(* PLC project EPEC_CU2.project, CODESYS V3.5 SP19, author XXXX *)
(* stored: creationDateTime 2026-03-19T14:01:24.5297586+02:00, modificationDateTime 2026-03-19T14:01:24.5297586+02:00, organization XXXX *)

(* NOTE! NOTE! NOTE! NOTE! NOTE! NOTE! NOTE! NOTE! NOTE! NOTE! NOTE! This object is created by Epec MultiTool. User changes are overwritten when project is imported. Content: - EventCode channel IDs *)
{attribute 'qualified_only'}
{attribute 'strict'}
TYPE ChannelIDs : (Ch1 := 0, Ch2, Ch3, Ch4) BYTE;
END_TYPE

(* NOTE! NOTE! NOTE! NOTE! NOTE! NOTE! NOTE! NOTE! NOTE! NOTE! NOTE! This object is created by Epec MultiTool. User changes are overwritten when project is imported. Content: - EventCode device IDs *)
{attribute 'qualified_only'}
{attribute 'strict'}
TYPE DeviceIDs : (VoltageInput := 0, DigitalInput, CurrentInput, ParameterValidation) BYTE;
END_TYPE

TYPE IdentityObject : STRUCT
  VendorId : DWORD := 0;  (* Vendor ID *)
  ProductCode : DWORD := 0;  (* Product code *)
  Revision : DWORD := 0;  (* Revision number *)
  SerialNumber : DWORD := 0;  (* Serial number for control unit *)
END_STRUCT;
END_TYPE

{attribute 'qualified_only'}
{attribute 'location' := '16#800'}
{attribute 'strict'}
TYPE InitCanProtocolStates : (INIT_CANOPEN_PROTOCOLS := 1, INIT_CANOPEN_OD := 2, INIT_CANOPEN_PDO := 3, INIT_CANOPEN_OD_SAVE := 4, INIT_CANOPEN_OD_REORG := 5, INIT_J1939 := 6, INIT_PROTOCOLS_DONE := 7);
END_TYPE

TYPE IdentityObject : STRUCT
  VendorId : DWORD := 0;  (* Vendor ID *)
  ProductCode : DWORD := 0;  (* Product code *)
  Revision : DWORD := 0;  (* Revision number *)
  SerialNumber : DWORD := 0;  (* Serial number for control unit *)
END_STRUCT;
END_TYPE

{attribute 'analysis' := '-43'}
VAR_GLOBAL CONSTANT  (* G_CONSTANTS - NOTE! NOTE! NOTE! NOTE! NOTE! NOTE! NOTE! NOTE! NOTE! NOTE! NOTE! This object is created by Epec MultiTool. User changes are overwritten when project is imported. Content: - Project specific constant definitions *)
  DIAG_MCU_TEMP_HIGH_LIMIT : DINT := 125;  (* Diagnostic limit constants *)
  DIAG_MCU_TEMP_LOW_LIMIT : DINT := -40;
  DIAG_MCU_TEMP_DELAY : UINT := 50;
  DIAG_PCB1_TEMP_HIGH_LIMIT : DINT := 125;
  DIAG_PCB1_TEMP_LOW_LIMIT : DINT := -45;
  DIAG_PCB1_TEMP_DELAY : UINT := 100;
  DIAG_PCB2_TEMP_HIGH_LIMIT : DINT := 105;
  DIAG_PCB2_TEMP_LOW_LIMIT : DINT := -40;
  DIAG_PCB2_TEMP_DELAY : UINT := 100;
  DIAG_SUPPLY_VOLTAGE_HIGH_LIMIT : DINT := 32000;
  DIAG_SUPPLY_VOLTAGE_LOW_LIMIT : DINT := 4500;
  DIAG_SUPPLY_VOLTAGE_DELAY : UINT := 450;
  DIAG_OUTPUT_GROUP1_HIGH_LIMIT : DINT := 37000;
  DIAG_OUTPUT_GROUP1_LOW_LIMIT : DINT := 4500;
  DIAG_OUTPUT_GROUP1_DELAY : UINT := 100;
  G_PARAMHANDLERKEYWORD : DWORD := 16#226D6F52;  (* Parameterhandler keyword *)
  G_PARAMETER_SAVE_STATUS_ERROR : BYTE := BYTE#16#00;
  G_PARAMETER_SAVE_STATUS_DONE : BYTE := BYTE#16#01;
  G_PARAMETER_SAVE_STATUS_IN_PROGRESS : BYTE := BYTE#16#FF;
  G_SAFE_PARAMETERS_AUTHENTICATED : BYTE := BYTE#1;
  G_SAFE_PARAMETERS_NOT_AUTHENTICATED : BYTE := BYTE#0;
END_VAR

{attribute 'qualified_only'}
VAR_GLOBAL  (* G_CAN - NOTE! NOTE! NOTE! NOTE! NOTE! NOTE! NOTE! NOTE! NOTE! NOTE! NOTE! This object is created by Epec MultiTool. User changes are overwritten when project is imported. Content: - CAN definitions *)
  Channel1 : EPEC_CANL2.Channel;
  Channel2 : EPEC_CANL2.Channel;
  Channel3 : EPEC_CANL2.Channel;
  Channel4 : EPEC_CANL2.Channel;
  Channel5 : EPEC_CANL2.Channel;
  Channel6 : EPEC_CANL2.Channel;
END_VAR

{attribute 'qualified_only'}
{attribute 'location' := '16#800'}
{attribute 'analysis' := '-6, -12, -33, -43'}
VAR_GLOBAL  (* G_Common *)
  ParHandler : EPEC_PH.ParameterHandler;  (* Parameterhandler. Utility library for ODSave. Library handles parameter image modification. *)
  ParameterArea : ARRAY[1..EPEC_HWD.LibParameters.G_PARAM_AREA_MAX_SIZE] OF BYTE;  (* Parameter image *)
  FastParHandler : EPEC_PH.ParameterHandler;
  FastParameterArea : ARRAY[1..EPEC_HWD.LibParameters.G_USER_VALUE_AREA_MAX_SIZE] OF BYTE;
  FastParameters : FastParameters;
  SaveFastParameters : BOOL := FALSE;
  ParhandlerDisableChanges : BOOL := FALSE;  (* Flag to call Parhandler.DisableChanges(TRUE) *)
  ParhandlerEnableChanges : BOOL := FALSE;  (* Flag to call Parhandler.DisableChanges(FALSE) *)
  CAN1SSDOHandlerGrantAccess : BOOL := FALSE;  (* Flag to call G_CANopen_CAN1.SSDO_Handler.GrantAccessToSafetyParameters(TRUE) *)
  CAN2SSDOHandlerGrantAccess : BOOL := FALSE;  (* Flag to call G_CANopen_CAN2.SSDO_Handler.GrantAccessToSafetyParameters(TRUE) *)
  CAN3SSDOHandlerGrantAccess : BOOL := FALSE;  (* Flag to call G_CANopen_CAN3.SSDO_Handler.GrantAccessToSafetyParameters(TRUE) *)
  CAN4SSDOHandlerGrantAccess : BOOL := FALSE;  (* Flag to call G_CANopen_CAN4.SSDO_Handler.GrantAccessToSafetyParameters(TRUE) *)
  CAN5SSDOHandlerGrantAccess : BOOL := FALSE;  (* Flag to call G_CANopen_CAN5.SSDO_Handler.GrantAccessToSafetyParameters(TRUE) *)
  CAN6SSDOHandlerGrantAccess : BOOL := FALSE;  (* Flag to call G_CANopen_CAN6.SSDO_Handler.GrantAccessToSafetyParameters(TRUE) *)
  ProjectKey : STRING(79) := 'KEeJGzzvbvqAy4c';  (* Project key, used for validating the response code *)
END_VAR


{attribute 'qualified_only'}
{attribute 'location' := '16#800'}
{attribute 'analysis' := '-6'}
VAR_GLOBAL  (* G_Logs *)
  ApplicationLog : EPEC_SERRLOG.ErrorLog;
  AppLogInitOK : BOOL;
END_VAR


{attribute 'qualified_only'}
{attribute 'location' := '16#800'}
{attribute 'analysis' := '-12, -33, -43'}
VAR_GLOBAL  (* G_StatusFlags - NOTE! NOTE! NOTE! NOTE! NOTE! NOTE! NOTE! NOTE! NOTE! NOTE! NOTE! This object is created by Epec MultiTool. User changes are overwritten when project is imported. Content: - PLC_PRG status flags *)
  CANopenCan1NMTResetRequest : BOOL := FALSE;  (* Reset request flags tell if module is wanted to reset after current application cycle. *)
  CANopenCan2NMTResetRequest : BOOL := FALSE;
  CANopenCan3NMTResetRequest : BOOL := FALSE;
  CANopenCan4NMTResetRequest : BOOL := FALSE;
  CANopenCan5NMTResetRequest : BOOL := FALSE;
  CANopenCan6NMTResetRequest : BOOL := FALSE;
  SystemOk : BOOL := FALSE;
  CustomLEDControlEnable : BOOL := FALSE;  (* Flags to control the status LED from the application *)
  RedLED : BOOL := FALSE;
  GreenLED : BOOL := FALSE;
  BlueLED : BOOL := FALSE;
  CustomLED2ControlEnable : BOOL := FALSE;  (* Flags to control the status LED 2 from the application *)
  RedLED2 : BOOL := FALSE;
  GreenLED2 : BOOL := FALSE;
  BlueLED2 : BOOL := FALSE;
END_VAR

{attribute 'qualified_only'}
VAR_GLOBAL  (* G_StatusFlags_Safe - NOTE! NOTE! NOTE! NOTE! NOTE! NOTE! NOTE! NOTE! NOTE! NOTE! NOTE! This object is created by Epec MultiTool. User changes are overwritten when project is imported. Content: - S_PLC_PRG status flags *)
  S_SafeOperationEnable : SAFEBOOL := FALSE;
END_VAR

{attribute 'qualified_only'}
{attribute 'location' := '16#800'}
{attribute 'analysis' := '-33, -43'}
VAR_GLOBAL  (* G_SystemInfo - NOTE! NOTE! NOTE! NOTE! NOTE! NOTE! NOTE! NOTE! NOTE! NOTE! NOTE! This object is created by Epec MultiTool. User changes are overwritten when project is imported. Content: - System information common for all ODs. *)
  ProjectInfo : PROJECT_INFO;
  DeviceName : STRING(79);  (* 16#1008: Manufacturer device name *)
  HWVersion : STRING(79);  (* 16#1009: Manufacturer hardware version *)
  SWVersion : STRING(79);  (* 16#100A: Manufacturer software version *)
  Identity : IdentityObject;  (* 16#1018: Identity object *)
  ToolsVersion : ARRAY[1..1] OF DWORD;  (* 16#2030 Codesys version *)
  WireHarnessId : ARRAY[1..30] OF WORD := [30(0)];  (* 16#2101 Wire harness Sub1: Wire harness ID enable Sub2: Wire harness ID internal adc config Sub3: Wire harness ID internal adc config Sub4: Wire harness ID internal adc config Sub5: Wire harness ID internal adc config Sub6: Wire harness ID internal adc config Sub7: Wire harness ID internal adc config Sub8: Wire harness ID internal adc config Sub9: Wire harness ID internal adc config Sub10: Wire harness ID internal adc config Sub11: Wire harness ID internal adc config Sub12: Wire harness ID internal adc config Sub13: Wire harness ID internal adc config Sub14: Wire harness ID internal adc config Sub15: Wire harness ID internal adc config Sub16: Wire harness ID internal adc config Sub17: Wire harness ID internal adc config Sub18: Wire harness ID internal adc config Sub19: Wire harness ID internal adc config Sub20: Wire harness ID internal adc config Sub21: Wire harness ID internal adc config Sub22: Wire harness ID internal adc config Sub23: Wire harness ID internal adc config Sub24: Wire harness ID internal adc config Sub25: Wire harness ID internal adc config Sub26: Wire harness ID default base offset Sub27: Wire harness ID calculated offset Sub28: Wire harness ID stored offset Sub29: Wire harness ID locked Sub30: Wire harness ID error *)
  SoftwareInformation : ARRAY[1..10] OF STRING(79) := [''];  (* 16#2130 Software information Sub1: Application version Sub2: Additional version information Sub3: Reserved for future use Sub4: Reserved for future use Sub5: Reserved for future use Sub6: Reserved for future use Sub7: Reserved for future use Sub8: Reserved for future use Sub9: Reserved for future use Sub10: Reserved for future use *)
  MACAddress : ARRAY[1..6] OF BYTE := [6(0)];  (* 16#2140 MAC address Sub1: MAC address byte 1 Sub2: MAC address byte 2 Sub3: MAC address byte 3 Sub4: MAC address byte 4 Sub5: MAC address byte 5 Sub6: MAC address byte 6 *)
  EthernetConfiguration : ARRAY[1..50] OF BYTE := [50(0)];  (* 16#2141 Ethernet configuration Sub1: Ethernet enabled/disabled Sub2: DHCP on/off Sub3: Reserved Sub4: Reserved Sub5: Reserved Sub6: Reserved Sub7: Reserved Sub8: Reserved Sub9: Reserved Sub10: Reserved Sub11: Reserved Sub12: Reserved Sub13: Reserved Sub14: Reserved Sub15: Reserved Sub16: Reserved Sub17: Reserved Sub18: Netstatus Sub19: IP address highest byte Sub20: IP address 3rd byte Sub21: IP address 2nd byte Sub22: IP address lowest byte Sub23: Gateway highest byte Sub24: Gateway 3rd byte Sub25: Gateway 2nd byte Sub26: Gateway lowest byte Sub27: Netmask highest byte Sub28: Netmask 3rd byte Sub29: Netmask 2nd byte Sub30: Netmask first byte Sub31: Reserved Sub32: Reserved Sub33: Reserved Sub34: Reserved Sub35: Reserved Sub36: Reserved Sub37: Reserved Sub38: Reserved Sub39: Reserved Sub40: Reserved Sub41: Reserved Sub42: Reserved Sub43: Reserved Sub44: Reserved Sub45: Reserved Sub46: Reserved Sub47: Reserved Sub48: Reserved Sub49: Reserved Sub50: Reserved *)
  CAN1_Comms : ARRAY[1..10] OF WORD := [10(0)];  (* 16#2150 CAN 1 Communication parameters Sub1: CODESYS communication enabled Sub2: CODESYS communication node-ID Sub3: Bit rate Sub4: Cable detection offset for CODESYS node-ID Sub5: Cable detection offset for PLCopen node-ID Sub6: Mask for cable detection pins Sub7: Reserved Sub8: Reserved Sub9: Reserved Sub10: PLCopen application node-ID in CAN1 *)
  CAN2_Comms : ARRAY[1..10] OF WORD := [10(0)];  (* 16#2151 CAN 2 Communication parameters Sub1: CODESYS communication enabled Sub2: CODESYS communication node-ID Sub3: Bit rate Sub4: Reserved Sub5: Reserved Sub6: Reserved Sub7: Reserved Sub8: Reserved Sub9: Reserved Sub10: PLCopen application node-ID in CAN2 *)
  CAN3_Comms : ARRAY[1..10] OF WORD := [10(0)];  (* 16#2152 CAN 3 Communication parameters Sub1: CODESYS communication enabled Sub2: CODESYS communication node-ID Sub3: Bit rate Sub4: Reserved Sub5: Reserved Sub6: Reserved Sub7: Reserved Sub8: Reserved Sub9: Reserved Sub10: PLCopen application node-ID in CAN3 *)
  CAN4_Comms : ARRAY[1..10] OF WORD := [10(0)];  (* 16#2153 CAN 4 Communication parameters Sub1: CODESYS communication enabled Sub2: CODESYS communication node-ID Sub3: Bit rate Sub4: Reserved Sub5: Reserved Sub6: Reserved Sub7: Reserved Sub8: Reserved Sub9: Reserved Sub10: PLCopen application node-ID in CAN4 *)
  CAN5_Comms : ARRAY[1..10] OF WORD := [10(0)];  (* 16#2154 CAN 5 Communication parameters Sub1: CODESYS communication enabled Sub2: CODESYS communication node-ID Sub3: Bit rate Sub4: Reserved Sub5: Reserved Sub6: Reserved Sub7: Reserved Sub8: Reserved Sub9: Reserved Sub10: PLCopen application node-ID in CAN5 *)
  CAN6_Comms : ARRAY[1..10] OF WORD := [10(0)];  (* 16#2155 CAN 6 Communication parameters Sub1: CODESYS communication enabled Sub2: CODESYS communication node-ID Sub3: Bit rate Sub4: Reserved Sub5: Reserved Sub6: Reserved Sub7: Reserved Sub8: Reserved Sub9: Reserved Sub10: PLCopen application node-ID in CAN6 *)
END_VAR

{attribute 'qualified_only'}
{attribute 'global_init_slot' := '49991'}
VAR_GLOBAL  (* G_CANopen_CAN1 - NOTE! NOTE! NOTE! NOTE! NOTE! NOTE! NOTE! NOTE! NOTE! NOTE! NOTE! This object is created by Epec MultiTool User changes are overwritten when project is imported Content - CANopen protocol variable definitions *)
  Device : EPEC_CANopen.Device;  (* CAN device *)
  OD : EPEC_CANopen.OD;  (* Object Dictionary data *)
  ODEntrys : ARRAY[1..86] OF EPEC_CANopen.ODEntry;
  Protocols : ARRAY[1..5] OF EPEC_CANopen.ProtocolEntry;  (* Protocol data *)
  HB : EPEC_CANopen.HBData;  (* Heartbeat producer/consumer protocol data *)
  HB_Handler : EPEC_CANopen.CANopenHB;  (* Heartbeat producer/consumer protocol handler *)
  NMT : EPEC_CANopen.NMTData;  (* NMT protocol data *)
  NMT_Handler : EPEC_CANopen.CANopenNMT;  (* NMT protocol handler *)
  SSDO : EPEC_CANopen.SSDOData;  (* SDO server protocol data *)
  SSDO_Handler : EPEC_CANopen.CANopenSDOServer;  (* SDO server protocol handler *)
  GFC : EPEC_CANopen.GFCData;  (* GFC protocol data *)
  GFC_Handler : EPEC_CANopen.CANopenGFC;  (* GFC protocol handler *)
  CSDOS : ARRAY[1..1] OF EPEC_CANopen.CANopenCSDO := [];  (* SDO client instances *)
  ConfigurationValidCallback : EPEC_CANopen.CallbackOfIndex13FEh;  (* 16#13FE Configuration valid *)
  AppLogDomain : EPEC_CANopen.Domain;  (* 16#2171 Application log domain *)
  SaveAll : EPEC_ODSave.SaveODSaveAll;
  DeleteAll : EPEC_ODSave.SaveODDeleteAll;
  SaveODHandler : EPEC_ODSave.SaveOD_Handler;
  SaveData : ARRAY[0..3] OF EPEC_ODSave.SaveODSubIndexDescription := [(StartIndex := 16#1000, EndIndex := 16#FFFF, GroupNum := 1), (StartIndex := 16#1000, EndIndex := 16#1FFF, GroupNum := 1), (StartIndex := 16#2000, EndIndex := 16#FFFF, GroupNum := 1), (StartIndex := 16#0, EndIndex := 16#0, GroupNum := 1)];
  SaveSubData1010h : EPEC_ODSave.SaveODSubService;
  OD_ReOrg : EPEC_CANopen.CANopenODReOrg;
END_VAR

{attribute 'qualified_only'}
{attribute 'location' := '16#800'}
{attribute 'global_init_slot' := '49990'}
VAR_GLOBAL  (* G_CANopen_CAN1_VAR - NOTE! NOTE! NOTE! NOTE! NOTE! NOTE! NOTE! NOTE! NOTE! NOTE! NOTE! This object is created by Epec MultiTool User changes are overwritten when project is imported Content - *)
  OD_Error : EPEC_CANopen.Errors := EPEC_CANopen.Errors.NotInitialized;
  ODSave_Error : EPEC_ODSave.SaveODErrors;
  Callback_Error : EPEC_CANopen.Errors := EPEC_CANopen.Errors.NotInitialized;
  ProtocolAdded : ARRAY[1..5] OF BOOL := [5(0)];
  HB_Error : EPEC_CANopen.Errors := EPEC_CANopen.Errors.NotInitialized;
  NMT_Error : EPEC_CANopen.Errors := EPEC_CANopen.Errors.NotInitialized;
  SSDO_Error : EPEC_CANopen.Errors := EPEC_CANopen.Errors.NotInitialized;
  GFC_Error : EPEC_CANopen.Errors := EPEC_CANopen.Errors.NotInitialized;
  GFC_Status : BYTE;  (* GFC status *)
  CSDO_Error : EPEC_CANopen.Errors := EPEC_CANopen.Errors.NotInitialized;
  OD_REORG_Error : EPEC_CANopen.Errors := EPEC_CANopen.Errors.NotInitialized;
  OdReOrgReady : BOOL := FALSE;  (* OD Reorganize operation ready *)
  ODSave_OperationReady : BOOL := FALSE;
  ODParametersInitialized : BOOL := FALSE;
  SaveSigns1010 : ARRAY[0..3] OF DWORD;
  InitProtocolsCanState : InitCanProtocolStates := InitCanProtocolStates.INIT_CANOPEN_PROTOCOLS;
END_VAR

{attribute 'qualified_only'}
{attribute 'location' := '16#800'}
{attribute 'analysis' := '-5, -6, -33, -43, -48'}
VAR_GLOBAL  (* G_CAN1_VAR - NOTE! NOTE! NOTE! NOTE! NOTE! NOTE! NOTE! NOTE! NOTE! NOTE! NOTE! This object is created by Epec MultiTool User changes are overwritten when project is imported Content - CANopen OD index data *)
  DeviceType_Device1 : UDINT := 405;  (* 16#1000 Information about the device type *)
  ErrorReg_Device1 : USINT := 0;  (* 16#1001 Error information *)
  ConfigurationValidStatus : BYTE := EPEC_CANopen.G_CANOPEN_SRD_CONF_INVALID;  (* 16#13FE SR Device configuration *)
  TPDO_DUMMY : BYTE := 0;  (* 16#2128 PDO Dummy Variable Index *)
  RPDO_DUMMY : BYTE := 0;  (* 16#2129 PDO Dummy Variable Index *)
  Parameter_CSV_unique_ID : UINT := 16#0000;  (* 16#2131 Parameter CSV unique ID *)
  NonSafetyParameterAuthenticationStatus : BYTE := 0;  (* 16#21EE Authentication status for non-safety parameter editing *)
  NonSafetyParameterPassword : STRING(79) := '';  (* 16#21EF Non-safety parameter password *)
  ParameterSaveStatus : BYTE := 0;  (* 16#21FA Parameter save information *)
  AuthenticationStatus : BYTE := G_CONSTANTS.G_SAFE_PARAMETERS_NOT_AUTHENTICATED;  (* 16#21FD Authentication information *)
  ChallengeCode : WORD := 0;  (* 16#21FE Challenge code for safety parameter editing *)
  ResponseCode : WORD := 0;  (* 16#21FF Response code for safety parameter editing *)
END_VAR

(* Tool version : '8.6.9547.24640' (MultiTool build version) Xml version : '1.0.0' (MultiTool xml file version) Control Unit : 'EPEC_CU2' (Name of the unit in MultiTool) Control Unit Type : 'CORE1_MCU-01-B-MCU' (Type of the unit in MultiTool, including the functional version) CODESYS Profile : 'CODESYS V3.5 SP19' (CODESYS profile that was selected in MultiTool) Device Description Version: '3.5.19.20' (Device description version that was selected in MultiTool) Export Time : '19.03.2026 14.01.24' (Date and time when exported from MultiTool) Export Path : 'C:\Codesys RPC\apps\CodesysRPC\EPEC_CU2' (Path where MultiTool exported) Project File : 'C:\Codesys RPC\apps\CodesysRPC\CodesysRPC.mtproject' (MultiTool project file name that was used) *)
{attribute 'analysis' := '-9'}
PROGRAM S_PLC_PRG
  VAR_OUTPUT
    o_InitDone : BOOL := FALSE;
  END_VAR

            
// Initialize application log
IF NOT G_Logs.AppLogInitOK THEN
	G_Logs.AppLogInitOK := EPEC_SERRLOG.S_InitErrorLog(i_pErrorLog:= ADR(G_Logs.ApplicationLog));
END_IF


(* PLC_PRG init must be done before S_PLC_PRG init *)
IF NOT o_InitDone AND PLC_PRG.o_InitDone THEN
	(* Code template safe FB initializations *)
	IF NOT S_Init_IO.o_Ready THEN
		S_Init_IO();
	ELSIF NOT EPEC_HWDIAG.S_CORE1MCU_Diagnostic.o_InitReady THEN
		EPEC_HWDIAG.S_CORE1MCU_Diagnostic.Init(
			S_i_SupplyVoltageHighLimit := G_CONSTANTS.DIAG_SUPPLY_VOLTAGE_HIGH_LIMIT,
			S_i_SupplyVoltageLowLimit := G_CONSTANTS.DIAG_SUPPLY_VOLTAGE_LOW_LIMIT,
			S_i_SupplyVoltageDiagDelay := G_CONSTANTS.DIAG_SUPPLY_VOLTAGE_DELAY,
			S_i_OutputGroup1HighVoltage := G_CONSTANTS.DIAG_OUTPUT_GROUP1_HIGH_LIMIT,
			S_i_OutputGroup1LowVoltage := G_CONSTANTS.DIAG_OUTPUT_GROUP1_LOW_LIMIT,
			S_i_OutputGroup1DiagDelay := G_CONSTANTS.DIAG_OUTPUT_GROUP1_DELAY,
			S_i_MCUTemperatureHighLimit := G_CONSTANTS.DIAG_MCU_TEMP_HIGH_LIMIT,
			S_i_MCUTemperatureLowLimit := G_CONSTANTS.DIAG_MCU_TEMP_LOW_LIMIT,
			S_i_MCUTemperatureDiagDelay := G_CONSTANTS.DIAG_MCU_TEMP_DELAY,
			S_i_PCB1TemperatureHighLimit := G_CONSTANTS.DIAG_PCB1_TEMP_HIGH_LIMIT,
			S_i_PCB1TemperatureLowLimit := G_CONSTANTS.DIAG_PCB1_TEMP_LOW_LIMIT,
			S_i_PCB1TemperatureDiagDelay := G_CONSTANTS.DIAG_PCB1_TEMP_DELAY,
			S_i_PCB2TemperatureHighLimit := G_CONSTANTS.DIAG_PCB2_TEMP_HIGH_LIMIT,
			S_i_PCB2TemperatureLowLimit := G_CONSTANTS.DIAG_PCB2_TEMP_LOW_LIMIT,
			S_i_PCB2TemperatureDiagDelay := G_CONSTANTS.DIAG_PCB2_TEMP_DELAY
		);

	ELSIF NOT S_Inputs.o_InitReady THEN
		S_Inputs(i_Initialize:=TRUE);
	ELSIF NOT S_Outputs.o_InitReady THEN
		S_Outputs(i_Initialize:=TRUE);

	ELSE
		(* User safe FB initialization *)
		S_MainInit(o_MainInitReady=>o_InitDone);	
	END_IF
	
(* Both safe and non-safe PRG's initializations must be finished
   before executing the programs. *)
ELSIF PLC_PRG.o_Initdone THEN
	(* Safe actions to execute before safe main program *)
	S_Inputs(i_Initialize:=FALSE);

	EPEC_HWDIAG.S_CORE1MCU_Diagnostic(
		i_SupplyVoltageInPin := S_Inputs.o_AI_VIN_V_Diagnostic,
		i_SupplyBeforeSafetySwitch1:= S_Inputs.o_AI_VIN_V_Diagnostic,
		i_SupplyAfterSafetySwitch1:= S_Inputs.o_AI_VOUT_SAFE_Diagnostic,
		i_MCUTemperature:= S_Inputs.o_AI_MCU_C_Diagnostic,
		i_PCBTemperatureChannel1:= S_Inputs.o_AI_PCB_1_V_Diagnostic,
		i_PCBTemperatureChannel2:= S_Inputs.o_AI_PCB_2_V_Diagnostic,
		i_CableDetectionSavedNodeId := TO_BYTE(G_SystemInfo.WireHarnessId[28]), // use stored offset as saved value
		i_CableDetectionDetectedNodeId := TO_BYTE(G_SystemInfo.WireHarnessId[27]) // use calculated offset as detected value
	);

	S_Outputs(i_Initialize:=FALSE, i_UpdateMeasurements:=TRUE);
	S_Safety_Status(i_Safe_InitDone:= o_InitDone,
					i_Nonsafe_InitDone:= PLC_PRG.o_InitDone,
					S_i_SafetySignaturesValid:= TRUE,				(* S_ValidateConfigurations does not exist *)
					S_i_SafetyParametersValid:= TRUE,				(* S_ValidateConfigurations does not exist *)
					S_o_SafeOperationEnable => G_StatusFlags_Safe.S_SafeOperationEnable);


	(* User safe main program *)
	S_Main();

	(* Safe actions to execute after safe main program *)
	S_Outputs(i_Initialize:=FALSE, i_UpdateMeasurements:=FALSE);


(* ELSE non-safe PLC_PRG initialization is not finished yet, do nothing *)
END_IF


              
          
END_PROGRAM

(* Tool version : '8.6.9547.24640' (MultiTool build version) Xml version : '1.0.0' (MultiTool xml file version) Control Unit : 'EPEC_CU2' (Name of the unit in MultiTool) Control Unit Type : 'CORE1_MCU-01-B-MCU' (Type of the unit in MultiTool, including the functional version) CODESYS Profile : 'CODESYS V3.5 SP19' (CODESYS profile that was selected in MultiTool) Device Description Version: '3.5.19.20' (Device description version that was selected in MultiTool) Export Time : '19.03.2026 14.01.24' (Date and time when exported from MultiTool) Export Path : 'C:\Codesys RPC\apps\CodesysRPC\EPEC_CU2' (Path where MultiTool exported) Project File : 'C:\Codesys RPC\apps\CodesysRPC\CodesysRPC.mtproject' (MultiTool project file name that was used) *)
{attribute 'location' := '16#800'}
PROGRAM PLC_PRG
  VAR_OUTPUT
    o_InitDone : BOOL := FALSE;
  END_VAR
  VAR
    ControlLED : EPEC_HWD.DiagnosticLEDWithIndex;
    ControlLED2 : EPEC_HWD.DiagnosticLEDWithIndex;
  END_VAR

            
IF NOT o_InitDone AND G_Logs.AppLogInitOK THEN

	(* Code template non-safe FB initializations *)
    IF NOT Init_Entry.o_Ready THEN
        Init_Entry();
    ELSIF NOT NVMemory.o_InitReady THEN
        NVMemory(i_Initialize:=TRUE);
	ELSIF NOT Init_CAN.o_Ready THEN
		Init_CAN();
	ELSIF NOT Init_CANopen_CAN1.o_Ready THEN
		Init_CANopen_CAN1();
	ELSIF NOT Init_CANopen_Parameters_OD1.o_Ready THEN
		Init_CANopen_Parameters_OD1();

    ELSE
        (* User non-safe initialization *)
        MainInit(o_MainInitReady=>o_InitDone);
    END_IF

(* Both safe and non-safe PRG's initializations must be finished
before executing the programs. *)
ELSIF S_PLC_PRG.o_InitDone THEN
    (* Non-safe actions to execute before non-safe main program *)
	G_CAN.Channel1.CheckMessages();
	G_CAN.Channel2.CheckMessages();
	G_CAN.Channel3.CheckMessages();
	G_CAN.Channel4.CheckMessages();
	G_CAN.Channel5.CheckMessages();
	G_CAN.Channel6.CheckMessages();
	Handle_CANopen_CAN1();

	Handle_Diagnostic();

	// Read latest firmware errors to application log when FW is in error state
	IF EPEC_HWDIAG.S_CORE1MCU_Diagnostic.S_o_FWDiagnosticTaskStatus = EPEC_IODRV.DIAGNOSTIC_TASK_STATUS.EDiagnosticStatusError THEN
		Handle_Firmware_Errors(i_ReadErrors:= TRUE);
	END_IF


    (* User non-safe main program *)
    Main();

    (* Non-safe actions to execute after non-safe main program *)

    NVMemory(i_Initialize:=FALSE);
(* ELSE safe S_PLC_PRG initialization is not finished yet, do nothing *)
END_IF

ControlLED(
	i_LEDIndex := 0,
	i_InitState := NOT PLC_PRG.o_Initdone OR NOT S_PLC_PRG.o_Initdone,
	i_ApplicationInSafeState := NOT EPEC_HWDIAG.S_CORE1MCU_Diagnostic.S_o_OutputGroup1Control,
	i_SystemOk := G_StatusFlags.SystemOk AND G_StatusFlags_Safe.S_SafeOperationEnable,
	i_CustomLEDControl := G_StatusFlags.CustomLEDControlEnable,
	i_RedLED := G_StatusFlags.RedLED,
	i_GreenLED := G_StatusFlags.GreenLED,
	i_BlueLED := G_StatusFlags.BlueLED,
	o_Error =>
);

// LED 2 is only controlled by application custom controls
IF G_StatusFlags.CustomLED2ControlEnable THEN
	ControlLED2(
		i_LEDIndex := 1,
		i_InitState := FALSE,
		i_ApplicationInSafeState := FALSE,
		i_SystemOk := FALSE,
		i_CustomLEDControl := G_StatusFlags.CustomLED2ControlEnable,
		i_RedLED := G_StatusFlags.RedLED2,
		i_GreenLED := G_StatusFlags.GreenLED2,
		i_BlueLED := G_StatusFlags.BlueLED2,
		o_Error =>
	);
END_IF

(* Call non-safe blocks that have been flagged from the safe program *)
IF G_Common.ParhandlerDisableChanges THEN
    G_Common.ParhandlerDisableChanges:=FALSE;
    G_Common.ParHandler.DisableChanges(TRUE);
END_IF

IF G_Common.ParhandlerEnableChanges THEN
    G_Common.ParhandlerEnableChanges:=FALSE;
    G_Common.ParHandler.DisableChanges(FALSE);
END_IF

IF G_Common.CAN1SSDOHandlerGrantAccess THEN
	G_Common.CAN1SSDOHandlerGrantAccess:= FALSE;
	G_CANopen_CAN1.SSDO_Handler.GrantAccessToSafetyParameters(TRUE);
	G_CANopen_CAN1.NMT.NmtState:= EPEC_CANopen.NMTState.Preoperational;
END_IF


              
          
END_PROGRAM

(* This PRG contains non safety-related code. The following attribute is autogenerated. Do not remove. *)
{attribute 'location' := '16#800'}
{attribute 'analysis' := '-9, -19'}
PROGRAM NVMemory
  VAR_INPUT
    i_Initialize : BOOL := TRUE;
  END_VAR
  VAR_OUTPUT
    o_InitReady : BOOL;
    o_InitError : BOOL;
    o_InputError : BOOL;
    o_ParameterBackupLoaded : BOOL;  (* Valid OD parameter backup image loaded during init. Note indication requires HWD lib 1.1.3.0. *)
    o_FastParameterBackupLoaded : BOOL;  (* Valid fast parameter backup image loaded during init. Note indication requires HWD lib 1.1.3.0. *)
    o_ODParameterError : EPEC_PH.ParamHandlerStatus := EPEC_PH.ParamHandlerStatus.NO_ERROR;
    o_FastParameterError : EPEC_PH.ParamHandlerStatus := EPEC_PH.ParamHandlerStatus.NO_ERROR;
    o_NVMemError : EPEC_SYSTEM.SYSTEM_ERROR_CODES := EPEC_SYSTEM.SYSTEM_ERROR_CODES.FW_ERR_OK;
    o_DM2Error : EPEC_PH.ParamHandlerStatus := EPEC_PH.ParamHandlerStatus.NO_ERROR;
    o_MachineTypeError : EPEC_PH.ParamHandlerStatus := EPEC_PH.ParamHandlerStatus.NO_ERROR;  (* Note indication requires HWD lib 1.1.5.0. *)
  END_VAR
  VAR
    parSaveBusy : BOOL := FALSE;
    parSaveDone : BOOL := FALSE;
    parSaveError : BOOL := FALSE;
    authenticated : BOOL := FALSE;
  END_VAR

            IF i_Initialize THEN
	EPEC_HWD.NVMem.SetParameterBackup(i_Enable := EPEC_HWD.LibParameters.G_PARAM_BACKUP_IN_USE);

	EPEC_HWD.NVMem.Init(
		i_NVMemoryIndex := 0,
		i_pParametersArea := ADR(G_Common.ParameterArea),
		i_ParameterAreaSize := TO_UDINT(SIZEOF(G_Common.ParameterArea)),
		i_pParameterHandler := ADR(G_Common.ParHandler),
		i_pUserValuesArea := ADR(G_Common.FastParameterArea),
		i_UserValueAreaSize := TO_UDINT(SIZEOF(G_Common.FastParameterArea)),
		i_pUserValueHandler := ADR(G_Common.FastParHandler),
		i_pUserValues := ADR(G_Common.FastParameters),
		i_UserValuesSize := SIZEOF(G_Common.FastParameters),
		i_pDM2Area := 0,
		i_DM2AreaSize := 0,
		i_pDM2Handler := 0,
		i_pMachineTypeArea := DWORD#0,
		i_MachineTypeAreaSize := UDINT#0,
		i_pMachineTypeHandler := DWORD#0,
		i_ParHandlerKeyword := G_CONSTANTS.G_PARAMHANDLERKEYWORD,
		o_InitReady => o_InitReady,
	);
	// Check if backup images were loaded during initialization
	IF o_InitReady THEN
		EPEC_HWD.NVMem.IsBackupLoaded(
			o_ParameterBackupLoaded => o_ParameterBackupLoaded,
			o_UserValueBackupLoaded => o_FastParameterBackupLoaded
		);
	END_IF
ELSE

	IF G_CAN1_VAR.AuthenticationStatus = G_CONSTANTS.G_SAFE_PARAMETERS_AUTHENTICATED THEN
		authenticated := TRUE;
	ELSE
		authenticated := FALSE;
	END_IF

	EPEC_HWD.NVMem(
		i_WriteParameters := G_Common.ParHandler.o_ParametersChanged,
		i_WriteUserValues := G_Common.SaveFastParameters,
		i_WriteDM2 := FALSE,
		i_WriteMachineType := FALSE,
		i_Authentication := authenticated,
		o_InitError => o_InitError,
		o_InputError => o_InputError,
		o_ParameterError => o_ODParameterError,
		o_UserValueError => o_FastParameterError,
		o_DM2Error => o_DM2Error,
		o_MachineTypeError => o_MachineTypeError,
		o_NVMemError => o_NVMemError,
		o_ParSaveBusy => parSaveBusy,
		o_ParSaveDone => parSaveDone,
		o_ParSaveError => parSaveError
	);

    (* Set parameter save status value *)
	IF parSaveBusy OR (NOT authenticated AND NOT G_CANopen_CAN1_VAR.ODSave_OperationReady) THEN
		G_CAN1_VAR.ParameterSaveStatus:= G_CONSTANTS.G_PARAMETER_SAVE_STATUS_IN_PROGRESS; 
	ELSIF parSaveDone THEN
		G_CAN1_VAR.ParameterSaveStatus:= G_CONSTANTS.G_PARAMETER_SAVE_STATUS_DONE; 
	ELSIF parSaveError THEN
		G_CAN1_VAR.ParameterSaveStatus:= G_CONSTANTS.G_PARAMETER_SAVE_STATUS_ERROR; 
	END_IF

	EPEC_SERRLOG.S_AddError_DWORD(i_ErrorCode:= ApplicationErrors.NVRAM_INIT, i_LibraryErrorCode:= BOOL_TO_DINT(o_InitError), i_Info1:= 0, i_Info2:= 0);
	EPEC_SERRLOG.S_AddError_DWORD(i_ErrorCode:= ApplicationErrors.NVRAM_INPUT, i_LibraryErrorCode:= BOOL_TO_DINT(o_InputError), i_Info1:= 0, i_Info2:= 0);
	EPEC_SERRLOG.S_AddError_DWORD(i_ErrorCode:= ApplicationErrors.NVRAM_FW, i_LibraryErrorCode:= o_NVMemError, i_Info1:= 0, i_Info2:= 0);
	EPEC_SERRLOG.S_AddError_DWORD(i_ErrorCode:= ApplicationErrors.NVRAM_OD, i_LibraryErrorCode:= INT_TO_DINT(o_ODParameterError), i_Info1:= 0, i_Info2:= 0);
	EPEC_SERRLOG.S_AddError_DWORD(i_ErrorCode:= ApplicationErrors.NVRAM_FASTPAR, i_LibraryErrorCode:= INT_TO_DINT(o_FastParameterError), i_Info1:= 0, i_Info2:= 0);
	EPEC_SERRLOG.S_AddError_DWORD(i_ErrorCode:= ApplicationErrors.NVRAM_MACHINETYPE, i_LibraryErrorCode:= INT_TO_DINT(o_MachineTypeError), i_Info1:= 0, i_Info2:= 0);


	(* User value save triggered, reset trigger *)
	G_Common.SaveFastParameters := FALSE;
END_IF
            
          
END_PROGRAM

(* NOTE! NOTE! NOTE! NOTE! NOTE! NOTE! NOTE! NOTE! NOTE! NOTE! NOTE! This object is created by Epec MultiTool User changes are overwritten when project is imported Content - Initialization of CAN channels This PRG contains non safety-related code. The following attribute is autogenerated. Do not remove. *)
{attribute 'location' := '16#800'}
{attribute 'analysis' := '-9, -38'}
PROGRAM Init_CAN
  VAR_OUTPUT
    o_Ready : BOOL := FALSE;
    o_Error : BOOL := FALSE;
    o_CAN1InitError : EPEC_CANVXD.ERROR := EPEC_CANVXD.ERROR.CHANNEL_NOT_INITIALIZED;
    o_CAN2InitError : EPEC_CANVXD.ERROR := EPEC_CANVXD.ERROR.CHANNEL_NOT_INITIALIZED;
    o_CAN3InitError : EPEC_CANVXD.ERROR := EPEC_CANVXD.ERROR.CHANNEL_NOT_INITIALIZED;
    o_CAN4InitError : EPEC_CANVXD.ERROR := EPEC_CANVXD.ERROR.CHANNEL_NOT_INITIALIZED;
    o_CAN5InitError : EPEC_CANVXD.ERROR := EPEC_CANVXD.ERROR.CHANNEL_NOT_INITIALIZED;
    o_CAN6InitError : EPEC_CANVXD.ERROR := EPEC_CANVXD.ERROR.CHANNEL_NOT_INITIALIZED;
  END_VAR

            o_CAN1InitError := G_CAN.Channel1.InitCAN(i_Channel := 0, i_BitRate := G_SystemInfo.CAN1_Comms[3], i_Flags := 0);
o_CAN2InitError := G_CAN.Channel2.InitCAN(i_Channel := 1, i_BitRate := EPEC_CANVXD.BITRATE_250K, i_Flags := 0);
o_CAN3InitError := G_CAN.Channel3.InitCAN(i_Channel := 2, i_BitRate := EPEC_CANVXD.BITRATE_250K, i_Flags := 0);
o_CAN4InitError := G_CAN.Channel4.InitCAN(i_Channel := 3, i_BitRate := EPEC_CANVXD.BITRATE_250K, i_Flags := 0);
o_CAN5InitError := G_CAN.Channel5.InitCAN(i_Channel := 4, i_BitRate := EPEC_CANVXD.BITRATE_250K, i_Flags := 0);
o_CAN6InitError := G_CAN.Channel6.InitCAN(i_Channel := 5, i_BitRate := EPEC_CANVXD.BITRATE_250K, i_Flags := 0);

IF EPEC_CANVXD.ERROR.NO_ERROR = o_CAN1InitError AND
	EPEC_CANVXD.ERROR.NO_ERROR = o_CAN2InitError AND
	EPEC_CANVXD.ERROR.NO_ERROR = o_CAN3InitError AND
	EPEC_CANVXD.ERROR.NO_ERROR = o_CAN4InitError AND
	EPEC_CANVXD.ERROR.NO_ERROR = o_CAN5InitError AND
	EPEC_CANVXD.ERROR.NO_ERROR = o_CAN6InitError THEN
	o_Error := FALSE;
ELSE
	o_Error := TRUE;

	EPEC_SERRLOG.S_AddError_DWORD(i_ErrorCode:= ApplicationErrors.CAN_INIT, i_LibraryErrorCode:= INT_TO_DINT(o_CAN1InitError), i_Info1:= 0, i_Info2:= 1);
	EPEC_SERRLOG.S_AddError_DWORD(i_ErrorCode:= ApplicationErrors.CAN_INIT, i_LibraryErrorCode:= INT_TO_DINT(o_CAN2InitError), i_Info1:= 0, i_Info2:= 2);
	EPEC_SERRLOG.S_AddError_DWORD(i_ErrorCode:= ApplicationErrors.CAN_INIT, i_LibraryErrorCode:= INT_TO_DINT(o_CAN3InitError), i_Info1:= 0, i_Info2:= 3);
	EPEC_SERRLOG.S_AddError_DWORD(i_ErrorCode:= ApplicationErrors.CAN_INIT, i_LibraryErrorCode:= INT_TO_DINT(o_CAN4InitError), i_Info1:= 0, i_Info2:= 4);
	EPEC_SERRLOG.S_AddError_DWORD(i_ErrorCode:= ApplicationErrors.CAN_INIT, i_LibraryErrorCode:= INT_TO_DINT(o_CAN5InitError), i_Info1:= 0, i_Info2:= 5);
	EPEC_SERRLOG.S_AddError_DWORD(i_ErrorCode:= ApplicationErrors.CAN_INIT, i_LibraryErrorCode:= INT_TO_DINT(o_CAN6InitError), i_Info1:= 0, i_Info2:= 6);
END_IF

o_Ready := TRUE;

          
END_PROGRAM

(* NOTE! NOTE! NOTE! NOTE! NOTE! NOTE! NOTE! NOTE! NOTE! NOTE! NOTE! This object is created by Epec MultiTool User changes are overwritten when project is imported Content - Set system information common for all ODs. This PRG contains non safety-related code. The following attribute is autogenerated. Do not remove. *)
{attribute 'location' := '16#800'}
{attribute 'analysis' := '-9, -19, -26'}
PROGRAM Init_Entry
  VAR_OUTPUT
    o_Ready : BOOL;
    o_PasswordChangeResult : EPEC_SYSTEM.SYSTEM_ERROR_CODES := EPEC_SYSTEM.SYSTEM_ERROR_CODES.FW_ERR_OK;
  END_VAR
  VAR
    CanNodeId : ARRAY [2..6] OF WORD;
    CanPLCopenNodeId : ARRAY [2..6] OF WORD;
    CanBitRate : ARRAY [2..6] OF WORD;
    ReadBytes : DWORD;
    RandomNumber : UDINT;
    SystemParameters : EPEC_HW.SystemParameters;
    PasswordType : BYTE;
    errorCode : EPEC_SYSTEM.SYSTEM_ERROR_CODES;
  END_VAR

            SystemParameters.ReadData();

/// 16#1008: Manufacturer device name
EPEC_SYSTEM.SystemParametersRead (16#1008,0,79,ADR(G_SystemInfo.DeviceName),ADR(ReadBytes));
 /// 16#1009: Manufacturer hardware version
EPEC_SYSTEM.SystemParametersRead (16#1009,0,79,ADR(G_SystemInfo.HWVersion),ADR(ReadBytes));
/// 16#100A: Manufacturer software version
G_SystemInfo.SWVersion := SystemParameters.o_SoftwareVersion;
/// 16#1018: Identity object 
G_SystemInfo.Identity.VendorId := SystemParameters.o_VendorId;          /// Vendor ID
G_SystemInfo.Identity.ProductCode := SystemParameters.o_ProductCode;    /// Product code
G_SystemInfo.Identity.Revision := SystemParameters.o_RevisionNumber;    /// Revision number
G_SystemInfo.Identity.SerialNumber := SystemParameters.o_SerialNumber;  /// Serial number for control unit
/// 16#2030 Codesys version
G_SystemInfo.ToolsVersion[1] := DWORD#50659328;
/// 16#2101 Wire harness ID
G_SystemInfo.WireHarnessId := SystemParameters.i_WireHarnessID;
/// 16#2141 MAC address
G_SystemInfo.MACAddress := SystemParameters.o_MAC;
/// 16#2141 Ethernet Communication parameters
G_SystemInfo.EthernetConfiguration := SystemParameters.i_Ethernet;
/// 16#2150 CAN 1 Communication parameters
G_SystemInfo.CAN1_Comms := SystemParameters.i_CAN1;

/// Read parameters for additional CANs from firmware
EPEC_SYSTEM.SystemParametersRead ((16#2151),2,2,ADR(CanNodeId[2]),ADR(ReadBytes));
EPEC_SYSTEM.SystemParametersRead ((16#2151),3,2,ADR(CanBitRate[2]),ADR(ReadBytes));
EPEC_SYSTEM.SystemParametersRead ((16#2151),10,2,ADR(CanPLCopenNodeId[2]),ADR(ReadBytes));
EPEC_SYSTEM.SystemParametersRead ((16#2152),2,2,ADR(CanNodeId[3]),ADR(ReadBytes));
EPEC_SYSTEM.SystemParametersRead ((16#2152),3,2,ADR(CanBitRate[3]),ADR(ReadBytes));
EPEC_SYSTEM.SystemParametersRead ((16#2152),10,2,ADR(CanPLCopenNodeId[3]),ADR(ReadBytes));
EPEC_SYSTEM.SystemParametersRead ((16#2153),2,2,ADR(CanNodeId[4]),ADR(ReadBytes));
EPEC_SYSTEM.SystemParametersRead ((16#2153),3,2,ADR(CanBitRate[4]),ADR(ReadBytes));
EPEC_SYSTEM.SystemParametersRead ((16#2153),10,2,ADR(CanPLCopenNodeId[4]),ADR(ReadBytes));
EPEC_SYSTEM.SystemParametersRead ((16#2154),2,2,ADR(CanNodeId[5]),ADR(ReadBytes));
EPEC_SYSTEM.SystemParametersRead ((16#2154),3,2,ADR(CanBitRate[5]),ADR(ReadBytes));
EPEC_SYSTEM.SystemParametersRead ((16#2154),10,2,ADR(CanPLCopenNodeId[5]),ADR(ReadBytes));
EPEC_SYSTEM.SystemParametersRead ((16#2155),2,2,ADR(CanNodeId[6]),ADR(ReadBytes));
EPEC_SYSTEM.SystemParametersRead ((16#2155),3,2,ADR(CanBitRate[6]),ADR(ReadBytes));
EPEC_SYSTEM.SystemParametersRead ((16#2155),10,2,ADR(CanPLCopenNodeId[6]),ADR(ReadBytes));
/// Set variables to communication arrays
G_SystemInfo.CAN2_Comms[2] := CanNodeId[2];
G_SystemInfo.CAN2_Comms[3] := CanBitRate[2];
G_SystemInfo.CAN2_Comms[10] := CanPLCopenNodeId[2];
G_SystemInfo.CAN3_Comms[2] := CanNodeId[3];
G_SystemInfo.CAN3_Comms[3] := CanBitRate[3];
G_SystemInfo.CAN3_Comms[10] := CanPLCopenNodeId[3];
G_SystemInfo.CAN4_Comms[2] := CanNodeId[4];
G_SystemInfo.CAN4_Comms[3] := CanBitRate[4];
G_SystemInfo.CAN4_Comms[10] := CanPLCopenNodeId[4];
G_SystemInfo.CAN5_Comms[2] := CanNodeId[5];
G_SystemInfo.CAN5_Comms[3] := CanBitRate[5];
G_SystemInfo.CAN5_Comms[10] := CanPLCopenNodeId[5];
G_SystemInfo.CAN6_Comms[2] := CanNodeId[6];
G_SystemInfo.CAN6_Comms[3] := CanBitRate[6];
G_SystemInfo.CAN6_Comms[10] := CanPLCopenNodeId[6];


/// Set user password if password is factory default
errorCode := EPEC_SYSTEM.SystemParametersRead(16#2032,2,1,ADR(PasswordType),ADR(ReadBytes));
IF(errorCode = EPEC_SYSTEM.SYSTEM_ERROR_CODES.FW_ERR_OK AND 0 = PasswordType) THEN
	o_PasswordChangeResult := EPEC_SYSTEM.PasswordUnlock(i_User := 'User', i_Password := '');
	IF(EPEC_SYSTEM.SYSTEM_ERROR_CODES.FW_ERR_OK = o_PasswordChangeResult) THEN
		o_PasswordChangeResult := EPEC_SYSTEM.PasswordChange('User', '', TO_STRING(G_SystemInfo.Identity.SerialNumber MOD 10000));
	END_IF
	IF(EPEC_SYSTEM.SYSTEM_ERROR_CODES.FW_ERR_OK = o_PasswordChangeResult) THEN
		o_PasswordChangeResult := EPEC_SYSTEM.SystemParametersSave();
	END_IF
END_IF

IF EPEC_SYSTEM.SYSTEM_ERROR_CODES.FW_ERR_OK = EPEC_SYSTEM.GetRandomNumber(o_rnd => RandomNumber) THEN
	G_CAN1_VAR.ChallengeCode:= UDINT_TO_WORD(RandomNumber);
	o_Ready:= TRUE;
ELSE
	o_Ready := FALSE;
END_IF

          
END_PROGRAM

(* NOTE! NOTE! NOTE! NOTE! NOTE! NOTE! NOTE! NOTE! NOTE! NOTE! NOTE! This object is created by Epec MultiTool User changes are overwritten when project is imported This PRG contains non safety-related code. The following attribute is autogenerated. Do not remove. *)
{attribute 'location' := '16#800'}
PROGRAM Init_CANopen_Parameters_OD1
  VAR_OUTPUT
    o_Ready : BOOL := FALSE;
  END_VAR

            G_CANopen_CAN1.SaveODHandler.InitializeODParams(i_Enable:=TRUE,
	o_Ready=>o_Ready,
	o_Error=>G_CANopen_CAN1_VAR.ODSave_Error);

          
END_PROGRAM

(* NOTE! NOTE! NOTE! NOTE! NOTE! NOTE! NOTE! NOTE! NOTE! NOTE! NOTE! This object is created by Epec MultiTool User changes are overwritten when project is imported Content - Non-safe system status update This PRG contains non safety-related code. The following attribute is autogenerated. Do not remove. *)
{attribute 'location' := '16#800'}
PROGRAM Handle_Diagnostic

            (* System Ok conditions *)
G_StatusFlags.SystemOk:=
		NOT Init_CAN.o_Error AND			(* No errors in bus init *)
		NOT Init_CANopen_CAN1.o_Error AND			(* No CANopen init errors *)
		NOT Handle_CANopen_CAN1.o_Error;


          
END_PROGRAM

(* NOTE! NOTE! NOTE! NOTE! NOTE! NOTE! NOTE! NOTE! NOTE! NOTE! NOTE! This object is created by Epec MultiTool User changes are overwritten when project is imported Content - Reads firmware error codes to application error log This PRG contains non safety-related code. The following attribute is autogenerated. Do not remove. *)
{attribute 'location' := '16#800'}
{attribute 'analysis' := '-9, -19'}
PROGRAM Handle_Firmware_Errors
  VAR_INPUT
    i_ReadErrors : BOOL;
  END_VAR
  VAR
    readErrorsOld : BOOL;
    fw_entries : ARRAY [1..EPEC_SERRLOG.LibParameters.G_ERROR_LOG_MAX_LINES] OF EPEC_SYSTEM.SystemLogEntry;
    return_code : EPEC_SYSTEM.SYSTEM_ERROR_CODES;
    lines_found : UDINT;
    i : UDINT;
    previous_time : UDINT;
    boot_detected : BOOL;
    fw_log_startupid : UDINT := UDINT#0;
    fw_log_startupid_exist : BOOL := FALSE;
    fw_log_startupid_size : DWORD;
  END_VAR

            IF i_ReadErrors AND NOT readErrorsOld THEN
	// Read FW log startup id value, if supported by FW
	return_code := EPEC_SYSTEM.SystemParametersRead(i_Index:=16#2039, i_SubIndex:=2, i_pBufferSize:=TO_DWORD(SIZEOF(fw_log_startupid)), i_pBuffer:=ADR(fw_log_startupid), i_pNbrOfReadByte:=ADR(fw_log_startupid_size));

	// Check if read was success
	IF return_code = EPEC_SYSTEM.SYSTEM_ERROR_CODES.FW_ERR_OK THEN
		fw_log_startupid_exist := TRUE;
	ELSE
		fw_log_startupid_exist := FALSE;
	END_IF

	// Read firmware errors
	return_code:= EPEC_SYSTEM.GetFWLogTail(
		i_count:= EPEC_SERRLOG.LibParameters.G_ERROR_LOG_MAX_LINES,
		i_logEntryArray:= ADR(fw_entries),
		o_found => lines_found
	);

	IF return_code = EPEC_SYSTEM.SYSTEM_ERROR_CODES.FW_ERR_OK AND lines_found > UDINT#0 THEN
		// Check if startup id is supported by FW
		IF fw_log_startupid_exist THEN
			// Add errors from buffer until startup id is found 
			FOR i:= 1 TO EPEC_SERRLOG.LibParameters.G_ERROR_LOG_MAX_LINES DO
				IF i <= lines_found AND fw_entries[i].Identifier >= fw_log_startupid THEN
					S_AddError_DWORD(
						i_ErrorCode:= ApplicationErrors.FW_ERROR,
						i_LibraryErrorCode:= fw_entries[i].Error,
						i_Info1:= fw_entries[i].Info,
						i_Info2:= fw_entries[i].Identifier);
				END_IF
			END_FOR
		ELSE
			// Add first error
			S_AddError_DWORD(
				i_ErrorCode:= ApplicationErrors.FW_ERROR,
				i_LibraryErrorCode:= fw_entries[1].Error,
				i_Info1:= fw_entries[1].Info,
				i_Info2:= fw_entries[1].Identifier);

			previous_time:= fw_entries[1].Timestamp;
			boot_detected:= FALSE;

			// Add errors until timestamp rollover is detected
			FOR i:= 2 TO EPEC_SERRLOG.LibParameters.G_ERROR_LOG_MAX_LINES DO
				IF i <= lines_found AND fw_entries[i].Timestamp <= previous_time AND NOT boot_detected THEN
					S_AddError_DWORD(
						i_ErrorCode:= ApplicationErrors.FW_ERROR,
						i_LibraryErrorCode:= fw_entries[i].Error,
						i_Info1:= fw_entries[i].Info,
						i_Info2:= fw_entries[i].Identifier);

					previous_time:= fw_entries[i].Timestamp;

				ELSIF fw_entries[i].Timestamp > previous_time THEN
					boot_detected := TRUE;
				END_IF
			END_FOR
		END_IF
	END_IF
END_IF
readErrorsOld:= i_ReadErrors;

          
END_PROGRAM

(* NOTE! NOTE! NOTE! NOTE! NOTE! NOTE! NOTE! NOTE! NOTE! NOTE! NOTE! This object is created by Epec MultiTool User changes are overwritten when project is imported Content - Safety status update. This PRG contains safety-related code. *)
{attribute 'analysis' := '-9, -130'}
PROGRAM S_Safety_Status
  VAR_INPUT
    i_Safe_InitDone : BOOL;
    i_Nonsafe_InitDone : BOOL;
    S_i_SafetySignaturesValid : SAFEBOOL;
    S_i_SafetyParametersValid : SAFEBOOL;
  END_VAR
  VAR_OUTPUT
    S_o_SafeOperationEnable : SAFEBOOL;
  END_VAR

            IF EPEC_HWDIAG.S_CORE1MCU_Diagnostic.S_o_DiagStatusOk AND (* System diagnostic ok*) 
    i_Safe_InitDone AND     (* Init has been executed successfully *) 
    i_Nonsafe_InitDone AND (*Non - safe init has been executed successfully *) 
    S_i_SafetySignaturesValid AND (*SRDO safety signatures are valid *) 
    S_i_SafetyParametersValid AND (*All safety parameters are valid *) 
    G_CANOPEN_GFC_VALID <> G_CANopen_CAN1_VAR.GFC_Status AND
	(* No CANopen protocol errors *)
	 NOT Init_CANopen_CAN1.o_Error
THEN
    S_o_SafeOperationEnable := TRUE;
    
ELSE 
    // Add error on falling edge
	IF S_o_SafeOperationEnable THEN
		EPEC_SERRLOG.S_AddError_DWORD(i_ErrorCode := ApplicationErrors.SAFE_OPERATION_DISABLED, i_LibraryErrorCode := EPEC_SERRLOG.LibConstants.G_ErrorNA, i_Info1:=0, i_Info2:=0);
	END_IF

	S_o_SafeOperationEnable := FALSE;
    
	// Check for CAN1 GFC activation
	EPEC_SERRLOG.S_AddError_DWORD(i_ErrorCode:=ApplicationErrors.GFC_STATUS, i_LibraryErrorCode:=BYTE_TO_DINT(G_CANopen_CAN1_VAR.GFC_Status), i_Info1:=0, i_Info2:=1);
    
	IF EPEC_HWDIAG.S_CORE1MCU_Diagnostic.o_DiagEnableStates.OutputGroup1_Diagnostic_Enable AND NOT EPEC_HWDIAG.S_CORE1MCU_Diagnostic.S_o_DiagStatusOk THEN
		// Trigger error if S_o_DiagStatusOk is not OK after output group diagnostic is enabled
		EPEC_SERRLOG.S_AddError_DWORD(
			i_ErrorCode := ApplicationErrors.HW_DIAGNOSTIC_FAULT,
			i_LibraryErrorCode := EPEC_SERRLOG.LibConstants.G_ErrorNA,
			i_Info1 := 0,
			i_Info2 := 0);
	END_IF
	// output group 1
	EPEC_SERRLOG.S_AddError_BYTE(
		i_ErrorCode := ApplicationErrors.HW_DIAG_OUT_PWR_GRP_1,
		i_LibraryErrorCode := EPEC_HWDIAG.S_CORE1MCU_Diagnostic.o_OutputGroup1Control_EC.EventID,
		i_Info1 := EPEC_HWDIAG.S_CORE1MCU_Diagnostic.o_OutputGroup1Control_EC.FunctionID,
		i_Info2 := EPEC_HWDIAG.S_CORE1MCU_Diagnostic.o_OutputGroup1Control_EC.DeviceID,
		i_Info3 := EPEC_HWDIAG.S_CORE1MCU_Diagnostic.o_OutputGroup1Control_EC.ChannelID,
		i_Info4 := 0,
		i_Info5 := 0,
		i_Info6 := 0,
		i_Info7 := 0,
		i_Info8 := 0);

	// supply voltage
	EPEC_SERRLOG.S_AddError_BYTE(
		i_ErrorCode := ApplicationErrors.HW_DIAG_IN_SUPPLY,
		i_LibraryErrorCode := EPEC_HWDIAG.S_CORE1MCU_Diagnostic.o_SupplyVoltage_EC.EventID,
		i_Info1 := EPEC_HWDIAG.S_CORE1MCU_Diagnostic.o_SupplyVoltage_EC.FunctionID,
		i_Info2 := EPEC_HWDIAG.S_CORE1MCU_Diagnostic.o_SupplyVoltage_EC.DeviceID,
		i_Info3 := EPEC_HWDIAG.S_CORE1MCU_Diagnostic.o_SupplyVoltage_EC.ChannelID,
		i_Info4 := 0,
		i_Info5 := 0,
		i_Info6 := 0,
		i_Info7 := 0,
		i_Info8 := 0);

	// MCU temperature
	EPEC_SERRLOG.S_AddError_BYTE(
		i_ErrorCode := ApplicationErrors.HW_DIAG_IN_MCU_TEMP,
		i_LibraryErrorCode := EPEC_HWDIAG.S_CORE1MCU_Diagnostic.o_MCUTemperatureEC.EventID,
		i_Info1 := EPEC_HWDIAG.S_CORE1MCU_Diagnostic.o_MCUTemperatureEC.FunctionID,
		i_Info2 := EPEC_HWDIAG.S_CORE1MCU_Diagnostic.o_MCUTemperatureEC.DeviceID,
		i_Info3 := EPEC_HWDIAG.S_CORE1MCU_Diagnostic.o_MCUTemperatureEC.ChannelID,
		i_Info4 := 0,
		i_Info5 := 0,
		i_Info6 := 0,
		i_Info7 := 0,
		i_Info8 := 0);

	// PCB temperature 1
	EPEC_SERRLOG.S_AddError_BYTE(
		i_ErrorCode := ApplicationErrors.HW_DIAG_IN_PCB_TEMP_1,
		i_LibraryErrorCode := EPEC_HWDIAG.S_CORE1MCU_Diagnostic.o_PCBTemperatureCh1_EC.EventID,
		i_Info1 := EPEC_HWDIAG.S_CORE1MCU_Diagnostic.o_PCBTemperatureCh1_EC.FunctionID,
		i_Info2 := EPEC_HWDIAG.S_CORE1MCU_Diagnostic.o_PCBTemperatureCh1_EC.DeviceID,
		i_Info3 := EPEC_HWDIAG.S_CORE1MCU_Diagnostic.o_PCBTemperatureCh1_EC.ChannelID,
		i_Info4 := 0,
		i_Info5 := 0,
		i_Info6 := 0,
		i_Info7 := 0,
		i_Info8 := 0);

	// PCB temperature 2
	EPEC_SERRLOG.S_AddError_BYTE(
		i_ErrorCode := ApplicationErrors.HW_DIAG_IN_PCB_TEMP_2,
		i_LibraryErrorCode := EPEC_HWDIAG.S_CORE1MCU_Diagnostic.o_PCBTemperatureCh2_EC.EventID,
		i_Info1 := EPEC_HWDIAG.S_CORE1MCU_Diagnostic.o_PCBTemperatureCh2_EC.FunctionID,
		i_Info2 := EPEC_HWDIAG.S_CORE1MCU_Diagnostic.o_PCBTemperatureCh2_EC.DeviceID,
		i_Info3 := EPEC_HWDIAG.S_CORE1MCU_Diagnostic.o_PCBTemperatureCh2_EC.ChannelID,
		i_Info4 := 0,
		i_Info5 := 0,
		i_Info6 := 0,
		i_Info7 := 0,
		i_Info8 := 0);


END_IF 
          
END_PROGRAM

(* NOTE! NOTE! NOTE! NOTE! NOTE! NOTE! NOTE! NOTE! NOTE! NOTE! NOTE! This object is created by Epec MultiTool User changes are overwritten when project is imported Content - CANopen initialization - Includes Init_CANopen_OD1 - CANopen data update This PRG contains non safety-related code. The following attribute is autogenerated. Do not remove. *)
{attribute 'location' := '16#800'}
{attribute 'analysis' := '-9, -19, -130'}
PROGRAM Init_CANopen_CAN1
  VAR_OUTPUT
    o_Ready : BOOL := FALSE;
    o_Error : BOOL := FALSE;
  END_VAR
  VAR
    odReOrgReady : BOOL := FALSE;
  END_VAR

            CASE G_CANopen_CAN1_VAR.InitProtocolsCanState OF

InitCanProtocolStates.INIT_CANOPEN_PROTOCOLS:
	G_CANopen_CAN1.Device.itfCanChannel:=G_CAN.Channel1; (*Connect device to can channel*)
	G_CANopen_CAN1.Device.NodeID := BYTE#4;
	G_CANopen_CAN1.NMT.NmtState:=EPEC_CANopen.NMTState.BootUp; (* Set NMT status to BOOTUP *)

	(*Initialize OD's data structures*)
	G_CANopen_CAN1.OD.EntryCount:=SIZEOF(G_CANopen_CAN1.ODEntrys)/SIZEOF(G_CANopen_CAN1.ODEntrys[1]); (*Max entries of given OD(CANopenDeviceODEntrys array)*)
	G_CANopen_CAN1.OD.InOrder:=FALSE; (*OD isn't in order*)
	G_CANopen_CAN1.OD.NextFree:=0; (*OD does not have any entries yet*)
	G_CANopen_CAN1.OD.pODEntry:=ADR(G_CANopen_CAN1.ODEntrys); (*Pointer to OD array*)

	(*Define NMT protocol*)
	G_CANopen_CAN1.Protocols[1].Protocol:=EPEC_CANopen.ProtocolType.NMT;
	G_CANopen_CAN1.Protocols[1].pData:=ADR(G_CANopen_CAN1.NMT);
	G_CANopen_CAN1.Protocols[1].itfProtocol:=G_CANopen_CAN1.NMT_Handler;
	G_CANopen_CAN1.Protocols[1].pError:=ADR(G_CANopen_CAN1_VAR.NMT_Error);
	G_CANopen_CAN1_VAR.ProtocolAdded[1] := CANopenDeviceAddProtocol( (* Add to protocol stack *)
		i_pDevice:=ADR(G_CANopen_CAN1.Device),
		i_pProtocol:=ADR(G_CANopen_CAN1.Protocols[1]),
	);

	(*Initialize NMT protocol*)
	IF G_CANopen_CAN1_VAR.ProtocolAdded[1] THEN
		G_CANopen_CAN1.NMT_Handler.Init(
			i_pDevice := ADR(G_CANopen_CAN1.Device),
			i_ThisIsMaster := FALSE,
			i_StartInterval :=  1000,
			i_pMonitoredNodes := 0,
			i_NumberOfNodes := 0,
			i_SimultaneousSlaveConfiguration := FALSE,
			i_pOdReOrg := ADR(G_CANopen_CAN1.OD_ReOrg),
			o_Error => G_CANopen_CAN1_VAR.NMT_Error
		);
	ELSE
		G_CANopen_CAN1_VAR.NMT_Error := EPEC_CANopen.Errors.ProtocolDataMissing;
	END_IF

	(*Define OD protocol*)
	G_CANopen_CAN1.Protocols[2].Protocol:=EPEC_CANopen.ProtocolType.OD;
	G_CANopen_CAN1.Protocols[2].pData:=ADR(G_CANopen_CAN1.OD);
	G_CANopen_CAN1.Protocols[2].pError:=ADR(G_CANopen_CAN1_VAR.OD_Error);
	G_CANopen_CAN1_VAR.ProtocolAdded[2] := CANopenDeviceAddProtocol( (* Add to protocol stack *)
		i_pDevice:=ADR(G_CANopen_CAN1.Device),
		i_pProtocol:=ADR(G_CANopen_CAN1.Protocols[2]),
	);
	IF NOT G_CANopen_CAN1_VAR.ProtocolAdded[2] THEN
		G_CANopen_CAN1_VAR.OD_Error := EPEC_CANopen.Errors.ProtocolDataMissing;
	END_IF

	(*Define HB protocol
	- Uses NMT and OD protocol data, thus need to be defined after them.
	*)
	G_CANopen_CAN1.HB.HeartBeat.PT := T#200MS; (* HB producer time *)

	G_CANopen_CAN1.Protocols[3].Protocol:=EPEC_CANopen.ProtocolType.HB;
	G_CANopen_CAN1.Protocols[3].pData:=ADR(G_CANopen_CAN1.HB);
	G_CANopen_CAN1.Protocols[3].itfProtocol:=G_CANopen_CAN1.HB_Handler;
	G_CANopen_CAN1.Protocols[3].pError:=ADR(G_CANopen_CAN1_VAR.HB_Error);
	G_CANopen_CAN1_VAR.ProtocolAdded[3] := CANopenDeviceAddProtocol( (* Add to protocol stack *)
		i_pDevice:=ADR(G_CANopen_CAN1.Device),
		i_pProtocol:=ADR(G_CANopen_CAN1.Protocols[3]),
	);

	(* Initialize HB protocol *)
	IF G_CANopen_CAN1_VAR.ProtocolAdded[3] THEN

		(* Add monitored nodes *)
		G_CANopen_CAN1.HB_Handler.Init(
			i_pDevice := ADR(G_CANopen_CAN1.Device),
			o_Error => G_CANopen_CAN1_VAR.HB_Error
		);
	ELSE
		G_CANopen_CAN1_VAR.HB_Error := EPEC_CANopen.Errors.ProtocolDataMissing;
	END_IF

	(*Define SSDO protocol*)
	G_CANopen_CAN1.Protocols[4].Protocol:=EPEC_CANopen.ProtocolType.SSDO;
	G_CANopen_CAN1.Protocols[4].pData:=ADR(G_CANopen_CAN1.SSDO);
	G_CANopen_CAN1.Protocols[4].itfProtocol:=G_CANopen_CAN1.SSDO_Handler;
	G_CANopen_CAN1.Protocols[4].pError:=ADR(G_CANopen_CAN1_VAR.SSDO_Error);
	G_CANopen_CAN1_VAR.ProtocolAdded[4] := CANopenDeviceAddProtocol( (* Add to protocol stack *)
		i_pDevice:=ADR(G_CANopen_CAN1.Device),
		i_pProtocol:=ADR(G_CANopen_CAN1.Protocols[4])
	);
	IF G_CANopen_CAN1_VAR.ProtocolAdded[4] THEN
		G_CANopen_CAN1.SSDO_Handler.Init(
			i_pDevice := ADR(G_CANopen_CAN1.Device),
			o_Error => G_CANopen_CAN1_VAR.SSDO_Error
		);
	ELSE
		G_CANopen_CAN1_VAR.SSDO_Error := EPEC_CANopen.Errors.ProtocolDataMissing;
	END_IF

	(*Define GFC protocol*)
	G_CANopen_CAN1.Protocols[5].Protocol:=EPEC_CANopen.ProtocolType.GFC;
	G_CANopen_CAN1.Protocols[5].pData:=ADR(G_CANopen_CAN1.GFC);
	G_CANopen_CAN1.Protocols[5].itfProtocol:=G_CANopen_CAN1.GFC_Handler;
	G_CANopen_CAN1.Protocols[5].pError:=ADR(G_CANopen_CAN1_VAR.GFC_Error);
	G_CANopen_CAN1_VAR.ProtocolAdded[5] := CANopenDeviceAddProtocol(  (* Add to protocol stack *)
		i_pDevice:=ADR(G_CANopen_CAN1.Device),
		i_pProtocol:=ADR(G_CANopen_CAN1.Protocols[5])
	);
	IF G_CANopen_CAN1_VAR.ProtocolAdded[5] THEN
		G_CANopen_CAN1.GFC_Handler.Init(
			i_pDevice := ADR(G_CANopen_CAN1.Device),
			i_pStatus:=ADR(G_CANopen_CAN1_VAR.GFC_Status),
			o_Error => G_CANopen_CAN1_VAR.GFC_Error
		);
	ELSE
		G_CANopen_CAN1_VAR.GFC_Error := EPEC_CANopen.Errors.ProtocolDataMissing;
	END_IF

	(* Init CSDO instance array for bus *)
	EPEC_CANopen.CANopenSDOManager.Init(
		i_pDevice:=ADR(G_CANopen_CAN1.Device),
		i_pCSDOArrayStart:=ADR(G_CANopen_CAN1.CSDOS),
		i_CSDOArraySize:=SIZEOF(G_CANopen_CAN1.CSDOS)/SIZEOF(G_CANopen_CAN1.CSDOS[1]),
		o_Error=>G_CANopen_CAN1_VAR.CSDO_Error
	);

	G_CANopen_CAN1_VAR.InitProtocolsCanState := InitCanProtocolStates.INIT_CANOPEN_OD;

InitCanProtocolStates.INIT_CANOPEN_OD:

	(* Add index data to OD *)
	Init_CANopen_OD1(o_Ready=>); (* Must be done before initing PDOs and SRDOs. *)

	IF Init_CANopen_OD1.o_Ready THEN
		G_CANopen_CAN1_VAR.InitProtocolsCanState := InitCanProtocolStates.INIT_CANOPEN_OD_SAVE;
	END_IF


InitCanProtocolStates.INIT_CANOPEN_OD_SAVE:

	(*Initialize OD save*)
	G_CANopen_CAN1.SaveSubData1010h.pSaveSigns := ADR(G_CANopen_CAN1_VAR.SaveSigns1010[0]);
	G_CANopen_CAN1.SaveSubData1010h.NumOfEntrys := 4;
	G_CANopen_CAN1.SaveSubData1010h.pSaveIndexData := ADR(G_CANopen_CAN1.SaveData[0]);
	G_CANopen_CAN1.SaveData[3].itfSaveAll := G_CANopen_CAN1.SaveAll;
	G_CANopen_CAN1.SaveData[3].itfDeleteAll := G_CANopen_CAN1.DeleteAll;
	G_CANopen_CAN1.OD.pAdditionalData := ADR(G_CANopen_CAN1.SaveSubData1010h);

	IF G_CANopen_CAN1_VAR.OD_Error = EPEC_CANopen.Errors.NoError THEN
		G_CANopen_CAN1.SaveODHandler.Init(
			i_pOD:= ADR(G_CANopen_CAN1.OD),
			i_pSaveAll:= ADR(G_CANopen_CAN1.SaveAll),
			i_pDeleteAll:= ADR(G_CANopen_CAN1.DeleteAll),
			i_pParamHandler:= ADR(G_Common.ParHandler),
			i_NumOfParamsPerCycle:= 50,
			o_Error => G_CANopen_CAN1_VAR.ODSave_Error);
	END_IF

	G_CANopen_CAN1.OD_ReOrg.Init(i_pOD := ADR(G_CANopen_CAN1.OD), i_NumOfODIndexPerCycle := 50);
	G_CANopen_CAN1.OD_ReOrg.Start();

	G_CANopen_CAN1_VAR.InitProtocolsCanState := InitCanProtocolStates.INIT_CANOPEN_OD_REORG;

InitCanProtocolStates.INIT_CANOPEN_OD_REORG:

	G_CANopen_CAN1.OD_ReOrg.Update(o_Ready => odReOrgReady, o_Error => G_CANopen_CAN1_VAR.OD_REORG_Error);

	IF odReOrgReady THEN
		(* Check all protocol init status flags *)
		IF G_CANopen_CAN1_VAR.NMT_Error = EPEC_CANopen.Errors.NoError AND
			G_CANopen_CAN1_VAR.SSDO_Error = EPEC_CANopen.Errors.NoError AND
			G_CANopen_CAN1_VAR.OD_Error = EPEC_CANopen.Errors.NoError AND
			G_CANopen_CAN1_VAR.HB_Error = EPEC_CANopen.Errors.NoError AND
			G_CANopen_CAN1_VAR.CSDO_Error = EPEC_CANopen.Errors.NoError AND
			G_CANopen_CAN1_VAR.GFC_Error = EPEC_CANopen.Errors.NoError AND
			G_CANopen_CAN1_VAR.OD_REORG_Error = EPEC_CANopen.Errors.NoError
		THEN
			o_Error := FALSE; (* No errors in protocol inits *)
		ELSE
			o_Error := TRUE;

			EPEC_SERRLOG.S_AddError_DWORD(i_ErrorCode:= ApplicationErrors.CANOPEN_INIT_NMT, i_LibraryErrorCode:= INT_TO_DINT(G_CANopen_CAN1_VAR.NMT_Error), i_Info1:= 0, i_Info2:= 1);
			EPEC_SERRLOG.S_AddError_DWORD(i_ErrorCode:= ApplicationErrors.CANOPEN_INIT_SSDO, i_LibraryErrorCode:= INT_TO_DINT(G_CANopen_CAN1_VAR.SSDO_Error), i_Info1:= 0, i_Info2:= 1);
			EPEC_SERRLOG.S_AddError_DWORD(i_ErrorCode:= ApplicationErrors.CANOPEN_INIT_OD, i_LibraryErrorCode:= INT_TO_DINT(G_CANopen_CAN1_VAR.OD_Error), i_Info1:= 0, i_Info2:= 1);
			EPEC_SERRLOG.S_AddError_DWORD(i_ErrorCode:= ApplicationErrors.CANOPEN_INIT_HB, i_LibraryErrorCode:= INT_TO_DINT(G_CANopen_CAN1_VAR.HB_Error), i_Info1:= 0, i_Info2:= 1);
			EPEC_SERRLOG.S_AddError_DWORD(i_ErrorCode:= ApplicationErrors.CANOPEN_INIT_CSDO, i_LibraryErrorCode:= INT_TO_DINT(G_CANopen_CAN1_VAR.CSDO_Error), i_Info1:= 0, i_Info2:= 1);
			EPEC_SERRLOG.S_AddError_DWORD(i_ErrorCode:= ApplicationErrors.CANOPEN_INIT_GFC, i_LibraryErrorCode:= INT_TO_DINT(G_CANopen_CAN1_VAR.GFC_Error), i_Info1:= 0, i_Info2:= 1);
			EPEC_SERRLOG.S_AddError_DWORD(i_ErrorCode:= ApplicationErrors.CANOPEN_INIT_OD_REORG, i_LibraryErrorCode:= INT_TO_DINT(G_CANopen_CAN1_VAR.OD_REORG_Error), i_Info1:= 0, i_Info2:= 1);

		END_IF

		o_Ready:=TRUE;
		G_CANopen_CAN1_VAR.InitProtocolsCanState := InitCanProtocolStates.INIT_PROTOCOLS_DONE;
	END_IF
END_CASE

          
END_PROGRAM

(* NOTE! NOTE! NOTE! NOTE! NOTE! NOTE! NOTE! NOTE! NOTE! NOTE! NOTE! This object is created by Epec MultiTool User changes are overwritten when project is imported Content - CANopen object dictionary initialization This PRG contains non safety-related code. The following attribute is autogenerated. Do not remove. *)
{attribute 'location' := '16#800'}
{attribute 'analysis' := '-19'}
PROGRAM Init_CANopen_OD1
  VAR_OUTPUT
    o_Ready : BOOL := FALSE;
  END_VAR

            CASE G_CANopen_CAN1_VAR.InitProtocolsCanState OF

InitCanProtocolStates.INIT_CANOPEN_OD:

	(*16#0001..16#0009 Default types *)
	G_CANopen_CAN1_VAR.OD_Error := EPEC_CANopen.CANopenODAddDefautTypes(
		i_pOD:= ADR(G_CANopen_CAN1.OD)
	);

	(* 16#1000 Information about the device type *)
	IF G_CANopen_CAN1_VAR.OD_Error = EPEC_CANopen.Errors.NoError THEN
		G_CANopen_CAN1_VAR.OD_Error := CANopenODAddLine(
			i_pOD := ADR(G_CANopen_CAN1.OD),(*Address of Object dictionary where index will be added*)
			i_Index := G_CANOPEN_ODINDEX_DEVICE_TYPE,
			i_ObjectCode := EPEC_CANopen.ObjectCode.OD_VAR,(*Type of index*)
			i_NumOfSubids := USINT#0,(*Number of subindexes*)
			i_TypeSpec := EPEC_CANopen.DataType.Deftype_UNSIGNED32,(*Index datatype, either user defined or standard CiA 301*)
			i_ObjectAccess := G_CANOPEN_OD_ACCESS_NOWRITE OR G_CANOPEN_OD_ACCESS_SUB0NOWRITE,
			i_Sub0data := USINT#0,(*Value of subindex0 in array or (def)struct*)
			i_pIndexData := ADR(G_CAN1_VAR.DeviceType_Device1),
			i_itfSDOHandler := DWORD#0
		);
	END_IF

	(* 16#1001 Error information *)
	IF G_CANopen_CAN1_VAR.OD_Error = EPEC_CANopen.Errors.NoError THEN
		G_CANopen_CAN1_VAR.OD_Error := CANopenODAddLine(
			i_pOD := ADR(G_CANopen_CAN1.OD),(*Address of Object dictionary where index will be added*)
			i_Index := G_CANOPEN_ODINDEX_ERROR_REGISTER,
			i_ObjectCode := EPEC_CANopen.ObjectCode.OD_VAR,(*Type of index*)
			i_NumOfSubids := USINT#0,(*Number of subindexes*)
			i_TypeSpec := EPEC_CANopen.DataType.Deftype_UNSIGNED8,(*Index datatype, either user defined or standard CiA 301*)
			i_ObjectAccess := G_CANOPEN_OD_ACCESS_NOWRITE OR G_CANOPEN_OD_ACCESS_SUB0NOWRITE,
			i_Sub0data := USINT#0,(*Value of subindex0 in array or (def)struct*)
			i_pIndexData := ADR(G_CAN1_VAR.ErrorReg_Device1),
			i_itfSDOHandler := DWORD#0
		);
	END_IF

	(* 16#1008 Manufacturer device name *)
	IF G_CANopen_CAN1_VAR.OD_Error = EPEC_CANopen.Errors.NoError THEN
		G_CANopen_CAN1_VAR.OD_Error := CANopenODAddLine(
			i_pOD := ADR(G_CANopen_CAN1.OD),(*Address of Object dictionary where index will be added*)
			i_Index := G_CANOPEN_ODINDEX_MF_DEVICE_NAME,
			i_ObjectCode := EPEC_CANopen.ObjectCode.OD_VAR,(*Type of index*)
			i_NumOfSubids := USINT#0,(*Number of subindexes*)
			i_TypeSpec := EPEC_CANopen.DataType.Deftype_STRING,(*Index datatype, either user defined or standard CiA 301*)
			i_ObjectAccess := G_CANOPEN_OD_ACCESS_NOWRITE OR G_CANOPEN_OD_ACCESS_SUB0NOWRITE,
			i_Sub0data := USINT#0,(*Value of subindex0 in array or (def)struct*)
			i_pIndexData := ADR(G_SystemInfo.DeviceName),
			i_itfSDOHandler := DWORD#0
		);
	END_IF

	(* 16#1009 Hardware name *)
	IF G_CANopen_CAN1_VAR.OD_Error = EPEC_CANopen.Errors.NoError THEN
		G_CANopen_CAN1_VAR.OD_Error := CANopenODAddLine(
			i_pOD := ADR(G_CANopen_CAN1.OD),(*Address of Object dictionary where index will be added*)
			i_Index := G_CANOPEN_ODINDEX_MF_HW_VERSION,
			i_ObjectCode := EPEC_CANopen.ObjectCode.OD_VAR,(*Type of index*)
			i_NumOfSubids := USINT#0,(*Number of subindexes*)
			i_TypeSpec := EPEC_CANopen.DataType.Deftype_STRING,(*Index datatype, either user defined or standard CiA 301*)
			i_ObjectAccess := G_CANOPEN_OD_ACCESS_NOWRITE OR G_CANOPEN_OD_ACCESS_SUB0NOWRITE,
			i_Sub0data := USINT#0,(*Value of subindex0 in array or (def)struct*)
			i_pIndexData := ADR(G_SystemInfo.HWVersion),
			i_itfSDOHandler := DWORD#0
		);
	END_IF

	(* 16#100A Manufacturer software version *)
	IF G_CANopen_CAN1_VAR.OD_Error = EPEC_CANopen.Errors.NoError THEN
		G_CANopen_CAN1_VAR.OD_Error := CANopenODAddLine(
			i_pOD := ADR(G_CANopen_CAN1.OD),(*Address of Object dictionary where index will be added*)
			i_Index := G_CANOPEN_ODINDEX_MF_SW_VERSION,
			i_ObjectCode := EPEC_CANopen.ObjectCode.OD_VAR,(*Type of index*)
			i_NumOfSubids := USINT#0,(*Number of subindexes*)
			i_TypeSpec := EPEC_CANopen.DataType.Deftype_STRING,(*Index datatype, either user defined or standard CiA 301*)
			i_ObjectAccess := G_CANOPEN_OD_ACCESS_NOWRITE OR G_CANOPEN_OD_ACCESS_SUB0NOWRITE,
			i_Sub0data := USINT#0,(*Value of subindex0 in array or (def)struct*)
			i_pIndexData := ADR(G_SystemInfo.SWVersion),
			i_itfSDOHandler := DWORD#0
		);
	END_IF

	(* 16#1018   Vendor ID *)
	IF G_CANopen_CAN1_VAR.OD_Error = EPEC_CANopen.Errors.NoError THEN
		G_CANopen_CAN1_VAR.OD_Error := CANopenODAddLine(
			i_pOD := ADR(G_CANopen_CAN1.OD),(*Address of Object dictionary where index will be added*)
			i_Index := G_CANOPEN_ODINDEX_IDENTITY_OBJECT,
			i_ObjectCode := EPEC_CANopen.ObjectCode.OD_ARRAY, (*Type of index*)
			i_NumOfSubids := USINT#4,(*Number of subindexes*)
			i_TypeSpec := EPEC_CANopen.DataType.Deftype_UNSIGNED32,(*Index of 16-bit deftype*)
			i_ObjectAccess := G_CANOPEN_OD_ACCESS_NOWRITE OR G_CANOPEN_OD_ACCESS_SUB0NOWRITE,
			i_Sub0data := USINT#4,(*Value of subindex0 in array or (def)struct*)
			i_pIndexData := ADR(G_SystemInfo.Identity),
			i_itfSDOHandler := DWORD#0
		);
	END_IF
(* 16#13FE   SR Device configuration valid status *)
IF G_CANopen_CAN1_VAR.OD_Error = EPEC_CANopen.Errors.NoError THEN
	G_CANopen_CAN1_VAR.OD_Error := CANopenODAddLine(
		i_pOD := ADR(G_CANopen_CAN1.OD),(*Address of Object dictionary where index will be added*)
		i_Index := G_CANOPEN_ODINDEX_CONFIGURATION_VALID,
		i_ObjectCode := EPEC_CANopen.ObjectCode.OD_VAR,(*Type of index*)
		i_NumOfSubids := USINT#0,(*Number of subindexes*)
		i_TypeSpec := EPEC_CANopen.DataType.Deftype_UNSIGNED8,(*Index datatype, either user defined or standard CiA 301*)
		i_ObjectAccess := G_CANOPEN_OD_ACCESS_READWRITE,
		i_Sub0data := BYTE#0,(*Value of subindex0 in array or (def)struct*)
		i_pIndexData := ADR(G_CAN1_VAR.ConfigurationValidStatus),
		i_itfSDOHandler := G_CANopen_CAN1.ConfigurationValidCallback
	);
END_IF

	(* 16#2030   CodesysVersion *)
	IF G_CANopen_CAN1_VAR.OD_Error = EPEC_CANopen.Errors.NoError THEN
		G_CANopen_CAN1_VAR.OD_Error := CANopenODAddLine(
			i_pOD := ADR(G_CANopen_CAN1.OD),(*Address of Object dictionary where index will be added*)
			i_Index := 16#2030,
			i_ObjectCode := EPEC_CANopen.ObjectCode.OD_ARRAY, (*Type of index*)
			i_NumOfSubids := USINT#1,(*Number of subindexes*)
			i_TypeSpec := EPEC_CANopen.DataType.Deftype_UNSIGNED32,(*Index of 16-bit deftype*)
			i_ObjectAccess := G_CANOPEN_OD_ACCESS_NOWRITE OR G_CANOPEN_OD_ACCESS_SUB0NOWRITE,
			i_Sub0data := USINT#1,(*Value of subindex0 in array or (def)struct*)
			i_pIndexData := ADR(G_SystemInfo.ToolsVersion),
			i_itfSDOHandler := DWORD#0
		);
	END_IF

	(* 16#2101   Wire harness ID enable *)
	IF G_CANopen_CAN1_VAR.OD_Error = EPEC_CANopen.Errors.NoError THEN
		G_CANopen_CAN1_VAR.OD_Error := CANopenODAddLine(
			i_pOD := ADR(G_CANopen_CAN1.OD),(*Address of Object dictionary where index will be added*)
			i_Index := 16#2101,
			i_ObjectCode := EPEC_CANopen.ObjectCode.OD_ARRAY, (*Type of index*)
			i_NumOfSubids := USINT#30,(*Number of subindexes*)
			i_TypeSpec := EPEC_CANopen.DataType.Deftype_UNSIGNED16,(*Index of 16-bit deftype*)
			i_ObjectAccess := G_CANOPEN_OD_ACCESS_NOWRITE OR G_CANOPEN_OD_ACCESS_SUB0NOWRITE,
			i_Sub0data := USINT#30,(*Value of subindex0 in array or (def)struct*)
			i_pIndexData := ADR(G_SystemInfo.WireHarnessId),
			i_itfSDOHandler := DWORD#0
		);
	END_IF

	(* 16#2128 PDO Dummy Variable Index *)
	IF G_CANopen_CAN1_VAR.OD_Error = EPEC_CANopen.Errors.NoError THEN
		G_CANopen_CAN1_VAR.OD_Error := CANopenODAddLine(
			i_pOD := ADR(G_CANopen_CAN1.OD),(*Address of Object dictionary where index will be added*)
			i_Index := 16#2128,
			i_ObjectCode := EPEC_CANopen.ObjectCode.OD_VAR,(*Type of index*)
			i_NumOfSubids := USINT#0,(*Number of subindexes*)
			i_TypeSpec := EPEC_CANopen.DataType.Deftype_UNSIGNED8,(*Index datatype, either user defined or standard CiA 301*)
			i_ObjectAccess := G_CANOPEN_OD_ACCESS_READWRITE,
			i_Sub0data := USINT#0,(*Value of subindex0 in array or (def)struct*)
			i_pIndexData := ADR(G_CAN1_VAR.TPDO_DUMMY),
			i_itfSDOHandler := DWORD#0
		);
	END_IF

	(* 16#2129 PDO Dummy Variable Index *)
	IF G_CANopen_CAN1_VAR.OD_Error = EPEC_CANopen.Errors.NoError THEN
		G_CANopen_CAN1_VAR.OD_Error := CANopenODAddLine(
			i_pOD := ADR(G_CANopen_CAN1.OD),(*Address of Object dictionary where index will be added*)
			i_Index := 16#2129,
			i_ObjectCode := EPEC_CANopen.ObjectCode.OD_VAR,(*Type of index*)
			i_NumOfSubids := USINT#0,(*Number of subindexes*)
			i_TypeSpec := EPEC_CANopen.DataType.Deftype_UNSIGNED8,(*Index datatype, either user defined or standard CiA 301*)
			i_ObjectAccess := G_CANOPEN_OD_ACCESS_READWRITE,
			i_Sub0data := USINT#0,(*Value of subindex0 in array or (def)struct*)
			i_pIndexData := ADR(G_CAN1_VAR.RPDO_DUMMY),
			i_itfSDOHandler := DWORD#0
		);
	END_IF

	(* 16#2130   Application version *)
	IF G_CANopen_CAN1_VAR.OD_Error = EPEC_CANopen.Errors.NoError THEN
		G_CANopen_CAN1_VAR.OD_Error := CANopenODAddLine(
			i_pOD := ADR(G_CANopen_CAN1.OD),(*Address of Object dictionary where index will be added*)
			i_Index := 16#2130,
			i_ObjectCode := EPEC_CANopen.ObjectCode.OD_ARRAY, (*Type of index*)
			i_NumOfSubids := USINT#10,(*Number of subindexes*)
			i_TypeSpec := EPEC_CANopen.DataType.Deftype_STRING,(*Index of 16-bit deftype*)
			i_ObjectAccess := G_CANOPEN_OD_ACCESS_NOWRITE OR G_CANOPEN_OD_ACCESS_SUB0NOWRITE,
			i_Sub0data := USINT#10,(*Value of subindex0 in array or (def)struct*)
			i_pIndexData := ADR(G_SystemInfo.SoftwareInformation),
			i_itfSDOHandler := DWORD#0
		);
	END_IF

	(* 16#2140   MAC address byte 1 *)
	IF G_CANopen_CAN1_VAR.OD_Error = EPEC_CANopen.Errors.NoError THEN
		G_CANopen_CAN1_VAR.OD_Error := CANopenODAddLine(
			i_pOD := ADR(G_CANopen_CAN1.OD),(*Address of Object dictionary where index will be added*)
			i_Index := 16#2140,
			i_ObjectCode := EPEC_CANopen.ObjectCode.OD_ARRAY, (*Type of index*)
			i_NumOfSubids := USINT#6,(*Number of subindexes*)
			i_TypeSpec := EPEC_CANopen.DataType.Deftype_UNSIGNED8,(*Index of 16-bit deftype*)
			i_ObjectAccess := G_CANOPEN_OD_ACCESS_NOWRITE OR G_CANOPEN_OD_ACCESS_SUB0NOWRITE,
			i_Sub0data := USINT#6,(*Value of subindex0 in array or (def)struct*)
			i_pIndexData := ADR(G_SystemInfo.MACAddress),
			i_itfSDOHandler := DWORD#0
		);
	END_IF

	(* 16#2141   Ethernet enabled/disabled *)
	IF G_CANopen_CAN1_VAR.OD_Error = EPEC_CANopen.Errors.NoError THEN
		G_CANopen_CAN1_VAR.OD_Error := CANopenODAddLine(
			i_pOD := ADR(G_CANopen_CAN1.OD),(*Address of Object dictionary where index will be added*)
			i_Index := 16#2141,
			i_ObjectCode := EPEC_CANopen.ObjectCode.OD_ARRAY, (*Type of index*)
			i_NumOfSubids := USINT#50,(*Number of subindexes*)
			i_TypeSpec := EPEC_CANopen.DataType.Deftype_UNSIGNED8,(*Index of 16-bit deftype*)
			i_ObjectAccess := G_CANOPEN_OD_ACCESS_READWRITE OR G_CANOPEN_OD_ACCESS_SUB0NOWRITE,
			i_Sub0data := USINT#50,(*Value of subindex0 in array or (def)struct*)
			i_pIndexData := ADR(G_SystemInfo.EthernetConfiguration),
			i_itfSDOHandler := DWORD#0
		);
	END_IF

	(* 16#2131 Parameter CSV unique ID *)
	IF G_CANopen_CAN1_VAR.OD_Error = EPEC_CANopen.Errors.NoError THEN
		G_CANopen_CAN1_VAR.OD_Error := CANopenODAddLine(
			i_pOD := ADR(G_CANopen_CAN1.OD),(*Address of Object dictionary where index will be added*)
			i_Index := 16#2131,
			i_ObjectCode := EPEC_CANopen.ObjectCode.OD_VAR,(*Type of index*)
			i_NumOfSubids := USINT#0,(*Number of subindexes*)
			i_TypeSpec := EPEC_CANopen.DataType.Deftype_UNSIGNED16,(*Index datatype, either user defined or standard CiA 301*)
			i_ObjectAccess := G_CANOPEN_OD_ACCESS_NOWRITE OR G_CANOPEN_OD_ACCESS_SUB0NOWRITE,
			i_Sub0data := USINT#0,(*Value of subindex0 in array or (def)struct*)
			i_pIndexData := ADR(G_CAN1_VAR.Parameter_CSV_unique_ID),
			i_itfSDOHandler := DWORD#0
		);
	END_IF

	(* 16#2150   CODESYS communication enabled *)
	IF G_CANopen_CAN1_VAR.OD_Error = EPEC_CANopen.Errors.NoError THEN
		G_CANopen_CAN1_VAR.OD_Error := CANopenODAddLine(
			i_pOD := ADR(G_CANopen_CAN1.OD),(*Address of Object dictionary where index will be added*)
			i_Index := 16#2150,
			i_ObjectCode := EPEC_CANopen.ObjectCode.OD_ARRAY, (*Type of index*)
			i_NumOfSubids := USINT#10,(*Number of subindexes*)
			i_TypeSpec := EPEC_CANopen.DataType.Deftype_UNSIGNED16,(*Index of 16-bit deftype*)
			i_ObjectAccess := G_CANOPEN_OD_ACCESS_READWRITE OR G_CANOPEN_OD_ACCESS_SUB0NOWRITE,
			i_Sub0data := USINT#10,(*Value of subindex0 in array or (def)struct*)
			i_pIndexData := ADR(G_SystemInfo.CAN1_Comms),
			i_itfSDOHandler := DWORD#0
		);
	END_IF

	(* 16#2151   CODESYS communication enabled *)
	IF G_CANopen_CAN1_VAR.OD_Error = EPEC_CANopen.Errors.NoError THEN
		G_CANopen_CAN1_VAR.OD_Error := CANopenODAddLine(
			i_pOD := ADR(G_CANopen_CAN1.OD),(*Address of Object dictionary where index will be added*)
			i_Index := 16#2151,
			i_ObjectCode := EPEC_CANopen.ObjectCode.OD_ARRAY, (*Type of index*)
			i_NumOfSubids := USINT#10,(*Number of subindexes*)
			i_TypeSpec := EPEC_CANopen.DataType.Deftype_UNSIGNED16,(*Index of 16-bit deftype*)
			i_ObjectAccess := G_CANOPEN_OD_ACCESS_READWRITE OR G_CANOPEN_OD_ACCESS_SUB0NOWRITE,
			i_Sub0data := USINT#10,(*Value of subindex0 in array or (def)struct*)
			i_pIndexData := ADR(G_SystemInfo.CAN2_Comms),
			i_itfSDOHandler := DWORD#0
		);
	END_IF

	(* 16#2152   CODESYS communication enabled *)
	IF G_CANopen_CAN1_VAR.OD_Error = EPEC_CANopen.Errors.NoError THEN
		G_CANopen_CAN1_VAR.OD_Error := CANopenODAddLine(
			i_pOD := ADR(G_CANopen_CAN1.OD),(*Address of Object dictionary where index will be added*)
			i_Index := 16#2152,
			i_ObjectCode := EPEC_CANopen.ObjectCode.OD_ARRAY, (*Type of index*)
			i_NumOfSubids := USINT#10,(*Number of subindexes*)
			i_TypeSpec := EPEC_CANopen.DataType.Deftype_UNSIGNED16,(*Index of 16-bit deftype*)
			i_ObjectAccess := G_CANOPEN_OD_ACCESS_READWRITE OR G_CANOPEN_OD_ACCESS_SUB0NOWRITE,
			i_Sub0data := USINT#10,(*Value of subindex0 in array or (def)struct*)
			i_pIndexData := ADR(G_SystemInfo.CAN3_Comms),
			i_itfSDOHandler := DWORD#0
		);
	END_IF

	(* 16#2153   CODESYS communication enabled *)
	IF G_CANopen_CAN1_VAR.OD_Error = EPEC_CANopen.Errors.NoError THEN
		G_CANopen_CAN1_VAR.OD_Error := CANopenODAddLine(
			i_pOD := ADR(G_CANopen_CAN1.OD),(*Address of Object dictionary where index will be added*)
			i_Index := 16#2153,
			i_ObjectCode := EPEC_CANopen.ObjectCode.OD_ARRAY, (*Type of index*)
			i_NumOfSubids := USINT#10,(*Number of subindexes*)
			i_TypeSpec := EPEC_CANopen.DataType.Deftype_UNSIGNED16,(*Index of 16-bit deftype*)
			i_ObjectAccess := G_CANOPEN_OD_ACCESS_READWRITE OR G_CANOPEN_OD_ACCESS_SUB0NOWRITE,
			i_Sub0data := USINT#10,(*Value of subindex0 in array or (def)struct*)
			i_pIndexData := ADR(G_SystemInfo.CAN4_Comms),
			i_itfSDOHandler := DWORD#0
		);
	END_IF

	(* 16#2154   CODESYS communication enabled *)
	IF G_CANopen_CAN1_VAR.OD_Error = EPEC_CANopen.Errors.NoError THEN
		G_CANopen_CAN1_VAR.OD_Error := CANopenODAddLine(
			i_pOD := ADR(G_CANopen_CAN1.OD),(*Address of Object dictionary where index will be added*)
			i_Index := 16#2154,
			i_ObjectCode := EPEC_CANopen.ObjectCode.OD_ARRAY, (*Type of index*)
			i_NumOfSubids := USINT#10,(*Number of subindexes*)
			i_TypeSpec := EPEC_CANopen.DataType.Deftype_UNSIGNED16,(*Index of 16-bit deftype*)
			i_ObjectAccess := G_CANOPEN_OD_ACCESS_READWRITE OR G_CANOPEN_OD_ACCESS_SUB0NOWRITE,
			i_Sub0data := USINT#10,(*Value of subindex0 in array or (def)struct*)
			i_pIndexData := ADR(G_SystemInfo.CAN5_Comms),
			i_itfSDOHandler := DWORD#0
		);
	END_IF

	(* 16#2155   CODESYS communication enabled *)
	IF G_CANopen_CAN1_VAR.OD_Error = EPEC_CANopen.Errors.NoError THEN
		G_CANopen_CAN1_VAR.OD_Error := CANopenODAddLine(
			i_pOD := ADR(G_CANopen_CAN1.OD),(*Address of Object dictionary where index will be added*)
			i_Index := 16#2155,
			i_ObjectCode := EPEC_CANopen.ObjectCode.OD_ARRAY, (*Type of index*)
			i_NumOfSubids := USINT#10,(*Number of subindexes*)
			i_TypeSpec := EPEC_CANopen.DataType.Deftype_UNSIGNED16,(*Index of 16-bit deftype*)
			i_ObjectAccess := G_CANOPEN_OD_ACCESS_READWRITE OR G_CANOPEN_OD_ACCESS_SUB0NOWRITE,
			i_Sub0data := USINT#10,(*Value of subindex0 in array or (def)struct*)
			i_pIndexData := ADR(G_SystemInfo.CAN6_Comms),
			i_itfSDOHandler := DWORD#0
		);
	END_IF

	(* 16#21EE Authentication status for non-safety parameter editing *)
	IF G_CANopen_CAN1_VAR.OD_Error = EPEC_CANopen.Errors.NoError THEN
		G_CANopen_CAN1_VAR.OD_Error := CANopenODAddLine(
			i_pOD := ADR(G_CANopen_CAN1.OD),(*Address of Object dictionary where index will be added*)
			i_Index := 16#21EE,
			i_ObjectCode := EPEC_CANopen.ObjectCode.OD_VAR,(*Type of index*)
			i_NumOfSubids := USINT#0,(*Number of subindexes*)
			i_TypeSpec := EPEC_CANopen.DataType.Deftype_UNSIGNED8,(*Index datatype, either user defined or standard CiA 301*)
			i_ObjectAccess := G_CANOPEN_OD_ACCESS_NOWRITE OR G_CANOPEN_OD_ACCESS_SUB0NOWRITE,
			i_Sub0data := USINT#0,(*Value of subindex0 in array or (def)struct*)
			i_pIndexData := ADR(G_CAN1_VAR.NonSafetyParameterAuthenticationStatus),
			i_itfSDOHandler := DWORD#0
		);
	END_IF

	(* 16#21EF Non-safety parameter password *)
	IF G_CANopen_CAN1_VAR.OD_Error = EPEC_CANopen.Errors.NoError THEN
		G_CANopen_CAN1_VAR.OD_Error := CANopenODAddLine(
			i_pOD := ADR(G_CANopen_CAN1.OD),(*Address of Object dictionary where index will be added*)
			i_Index := 16#21EF,
			i_ObjectCode := EPEC_CANopen.ObjectCode.OD_VAR,(*Type of index*)
			i_NumOfSubids := USINT#0,(*Number of subindexes*)
			i_TypeSpec := EPEC_CANopen.DataType.Deftype_STRING,(*Index datatype, either user defined or standard CiA 301*)
			i_ObjectAccess := G_CANOPEN_OD_ACCESS_SUB0NOREAD OR G_CANOPEN_OD_ACCESS_NOREAD,
			i_Sub0data := USINT#0,(*Value of subindex0 in array or (def)struct*)
			i_pIndexData := ADR(G_CAN1_VAR.NonSafetyParameterPassword),
			i_itfSDOHandler := DWORD#0
		);
	END_IF

	(* 16#21FD Authentication information *)
	IF G_CANopen_CAN1_VAR.OD_Error = EPEC_CANopen.Errors.NoError THEN
		G_CANopen_CAN1_VAR.OD_Error := CANopenODAddLine(
			i_pOD := ADR(G_CANopen_CAN1.OD),(*Address of Object dictionary where index will be added*)
			i_Index := 16#21FD,
			i_ObjectCode := EPEC_CANopen.ObjectCode.OD_VAR,(*Type of index*)
			i_NumOfSubids := USINT#0,(*Number of subindexes*)
			i_TypeSpec := EPEC_CANopen.DataType.Deftype_UNSIGNED8,(*Index datatype, either user defined or standard CiA 301*)
			i_ObjectAccess := G_CANOPEN_OD_ACCESS_NOWRITE OR G_CANOPEN_OD_ACCESS_SUB0NOWRITE,
			i_Sub0data := USINT#0,(*Value of subindex0 in array or (def)struct*)
			i_pIndexData := ADR(G_CAN1_VAR.AuthenticationStatus),
			i_itfSDOHandler := DWORD#0
		);
	END_IF

	(* 16#21FE Challenge code for safety parameter editing *)
	IF G_CANopen_CAN1_VAR.OD_Error = EPEC_CANopen.Errors.NoError THEN
		G_CANopen_CAN1_VAR.OD_Error := CANopenODAddLine(
			i_pOD := ADR(G_CANopen_CAN1.OD),(*Address of Object dictionary where index will be added*)
			i_Index := 16#21FE,
			i_ObjectCode := EPEC_CANopen.ObjectCode.OD_VAR,(*Type of index*)
			i_NumOfSubids := USINT#0,(*Number of subindexes*)
			i_TypeSpec := EPEC_CANopen.DataType.Deftype_UNSIGNED16,(*Index datatype, either user defined or standard CiA 301*)
			i_ObjectAccess := G_CANOPEN_OD_ACCESS_NOWRITE OR G_CANOPEN_OD_ACCESS_SUB0NOWRITE,
			i_Sub0data := USINT#0,(*Value of subindex0 in array or (def)struct*)
			i_pIndexData := ADR(G_CAN1_VAR.ChallengeCode),
			i_itfSDOHandler := DWORD#0
		);
	END_IF

	(* 16#21FF Response code for safety parameter editing *)
	IF G_CANopen_CAN1_VAR.OD_Error = EPEC_CANopen.Errors.NoError THEN
		G_CANopen_CAN1_VAR.OD_Error := CANopenODAddLine(
			i_pOD := ADR(G_CANopen_CAN1.OD),(*Address of Object dictionary where index will be added*)
			i_Index := 16#21FF,
			i_ObjectCode := EPEC_CANopen.ObjectCode.OD_VAR,(*Type of index*)
			i_NumOfSubids := USINT#0,(*Number of subindexes*)
			i_TypeSpec := EPEC_CANopen.DataType.Deftype_UNSIGNED16,(*Index datatype, either user defined or standard CiA 301*)
			i_ObjectAccess := G_CANOPEN_OD_ACCESS_SUB0NOREAD OR G_CANOPEN_OD_ACCESS_NOREAD,
			i_Sub0data := USINT#0,(*Value of subindex0 in array or (def)struct*)
			i_pIndexData := ADR(G_CAN1_VAR.ResponseCode),
			i_itfSDOHandler := DWORD#0
		);
	END_IF

	(*16#2170 Application log error count *)
	IF G_CANopen_CAN1_VAR.OD_Error = EPEC_CANopen.Errors.NoError THEN
		G_CANopen_CAN1_VAR.OD_Error := CANopenODAddLine(
			i_pOD:= ADR(G_CANopen_CAN1.OD), (*Address of Object dictionary where index will be added *)
			i_Index:= 16#2170,
			i_ObjectCode:= EPEC_CANopen.ObjectCode.OD_VAR, (*Type of index*)
			i_NumOfSubids:= USINT#0,(*Number of subindexes*)
			i_TypeSpec:= EPEC_CANopen.DataType.Deftype_UNSIGNED32,(*Index of 32 - bit deftype *)
			i_ObjectAccess:= G_CANOPEN_OD_ACCESS_NOWRITE OR G_CANOPEN_OD_ACCESS_SUB0NOWRITE,
			i_Sub0data := USINT#0,(*Value of subindex0 in array or (def)struct*)
			i_pIndexData:= ADR(G_Logs.ApplicationLog.count),
			i_itfSDOHandler:= DWORD#0
		);
	END_IF

	(*16#2171 Application log domain *)
		IF G_CANopen_CAN1_VAR.OD_Error = EPEC_CANopen.Errors.NoError THEN
		G_CANopen_CAN1.AppLogDomain.DataSize:= SIZEOF(G_Logs.ApplicationLog.loglines) * 8;
		G_CANopen_CAN1.AppLogDomain.pData:= ADR(G_Logs.ApplicationLog.loglines);

		G_CANopen_CAN1_VAR.OD_Error := CANopenODAddLine(
			i_pOD:= ADR(G_CANopen_CAN1.OD), (*Address of Object dictionary where index will be added *)
			i_Index:= 16#2171,
			i_ObjectCode:= EPEC_CANopen.ObjectCode.OD_DOMAIN, (*Type of index*)
			i_NumOfSubids:= USINT#0,(*Number of subindexes*)
			i_TypeSpec:= EPEC_CANopen.DataType.Deftype_Domain,(*Domain deftype *)
			i_ObjectAccess:= G_CANOPEN_OD_ACCESS_NOWRITE,
			i_Sub0data:= USINT#0,(*Value of subindex0 in array or (def)struct*)
			i_pIndexData:= ADR(G_CANopen_CAN1.AppLogDomain),
			i_itfSDOHandler:= DWORD#0
		);
	END_IF

	o_Ready := TRUE;
END_CASE

          
END_PROGRAM

(* NOTE! NOTE! NOTE! NOTE! NOTE! NOTE! NOTE! NOTE! NOTE! NOTE! NOTE! This object is created by Epec MultiTool User changes are overwritten when project is imported Content - CANopen data update This PRG contains non safety-related code. The following attribute is autogenerated. Do not remove. *)
{attribute 'location' := '16#800'}
{attribute 'analysis' := '-9, -169'}
PROGRAM Handle_CANopen_CAN1
  VAR_OUTPUT
    o_Error : BOOL := FALSE;
  END_VAR

            (* Update callback data *)
IF G_CAN.Channel1.GetLatestError() <> DWORD#0 THEN
	G_CANopen_CAN1_VAR.Callback_Error := EPEC_CANopen.Errors.CallbackError;
ELSE
	G_CANopen_CAN1_VAR.Callback_Error := EPEC_CANopen.Errors.NoError;
END_IF

(* Update protocol data *)
G_CANopen_CAN1.HB_Handler.Update(
	i_Enable := TRUE,
	o_Error => G_CANopen_CAN1_VAR.HB_Error
);
G_CANopen_CAN1.NMT_Handler.Update(
	i_Enable := TRUE,
	o_Error => G_CANopen_CAN1_VAR.NMT_Error
);
G_CANopen_CAN1.SSDO_Handler.Update(
	i_Enable := TRUE,
	o_Error => G_CANopen_CAN1_VAR.SSDO_Error
);
G_CANopen_CAN1.GFC_Handler.Update(
	i_Enable := TRUE,
	o_Error => G_CANopen_CAN1_VAR.GFC_Error
);

G_CANopen_CAN1.OD_ReOrg.Update(o_Ready => , o_Error => G_CANopen_CAN1_VAR.OD_REORG_Error);

G_CANopen_CAN1.SaveODHandler.Update(i_Enable := TRUE,
	o_Ready => G_CANopen_CAN1_VAR.ODSave_OperationReady,
	o_Error => G_CANopen_CAN1_VAR.ODSave_Error);

IF G_CANopen_CAN1_VAR.HB_Error = EPEC_CANopen.Errors.NoError AND
	G_CANopen_CAN1_VAR.NMT_Error = EPEC_CANopen.Errors.NoError AND
	G_CANopen_CAN1_VAR.SSDO_Error = EPEC_CANopen.Errors.NoError AND
	G_CANopen_CAN1_VAR.GFC_Error = EPEC_CANopen.Errors.NoError AND
	G_CANopen_CAN1_VAR.OD_REORG_Error = EPEC_CANopen.Errors.NoError
THEN
	o_Error := FALSE;
ELSE
	o_Error := TRUE;

	EPEC_SERRLOG.S_AddError_DWORD(i_ErrorCode:= ApplicationErrors.CANOPEN_UPDATE_HB, i_LibraryErrorCode:= INT_TO_DINT(G_CANopen_CAN1_VAR.HB_Error), i_Info1:= 0, i_Info2:= 1);
	EPEC_SERRLOG.S_AddError_DWORD(i_ErrorCode:= ApplicationErrors.CANOPEN_UPDATE_NMT, i_LibraryErrorCode:= INT_TO_DINT(G_CANopen_CAN1_VAR.NMT_Error), i_Info1:= 0, i_Info2:= 1);
	EPEC_SERRLOG.S_AddError_DWORD(i_ErrorCode:= ApplicationErrors.CANOPEN_UPDATE_SSDO, i_LibraryErrorCode:= INT_TO_DINT(G_CANopen_CAN1_VAR.SSDO_Error), i_Info1:= 0, i_Info2:= 1);
	EPEC_SERRLOG.S_AddError_DWORD(i_ErrorCode:= ApplicationErrors.CANOPEN_UPDATE_GFC, i_LibraryErrorCode:= INT_TO_DINT(G_CANopen_CAN1_VAR.GFC_Error), i_Info1:= 0, i_Info2:= 1);
	EPEC_SERRLOG.S_AddError_DWORD(i_ErrorCode:= ApplicationErrors.CANOPEN_UPDATE_OD_REORG, i_LibraryErrorCode:= INT_TO_DINT(G_CANopen_CAN1_VAR.OD_REORG_Error), i_Info1:= 0, i_Info2:= 1);

END_IF


(*Check for NMT reset *)
IF G_CANopen_CAN1.NMT.StateChanged THEN
	IF G_CANopen_CAN1.NMT.LastNmtCommand = EPEC_CANopen.NMTCommand.Reset OR
		G_CANopen_CAN1.NMT.LastNmtCommand = EPEC_CANopen.NMTCommand.ResetCommunication
	THEN
		(* If there is an NMT reset command for the IEC application CANopen device,
		   This is only informative, application decides how to react to the command *)
		G_StatusFlags.CANopenCan1NMTResetRequest := TRUE;
	END_IF
END_IF


          
END_PROGRAM

(* NOTE! NOTE! NOTE! NOTE! NOTE! NOTE! NOTE! NOTE! NOTE! NOTE! NOTE! This object is created by Epec MultiTool User changes are overwritten when project is imported Content - Init IO. This PRG contains safety-related code. The following attribute is autogenerated. Do not remove. *)
{attribute 'analysis' := '-9, -12'}
PROGRAM S_Init_IO
  VAR_OUTPUT
    o_Ready : SAFEBOOL := FALSE;
    o_Error : BOOL := FALSE;
    o_ErrorInConnector : DWORD := DWORD#0;
    o_ErrorInPin : DWORD := DWORD#0;
    o_FWErrorCode : EPEC_SYSTEM.SYSTEM_ERROR_CODES;
  END_VAR
  VAR
    result : EPEC_SYSTEM.SYSTEM_ERROR_CODES;
    pin : DWORD := DWORD#0;
    connector : DWORD := DWORD#0;
    info1 : DWORD := DWORD#0;  (* MSW connector, LSW pin *)
    info2 : DWORD := DWORD#0;  (* error specific *)
  END_VAR

            IF result = EPEC_SYSTEM.SYSTEM_ERROR_CODES.FW_ERR_OK THEN
	result := EPEC_IODRV.IoDrvSetState(EPEC_IODRV.IoDrvStates.IODRV_STATE_CONFIGURATION);
END_IF
(* Internal diagnostics *)
(* Init for I/O which are for diagnostic. *)

IF result = EPEC_SYSTEM.SYSTEM_ERROR_CODES.FW_ERR_OK THEN
	connector := 255; // internal
	pin := 1;
	result := EPEC_IODRV.IoDrvDISetMode(EPEC_HW.IO_Channels.PIN_1000_1_DI_FACTORY_RESET, EPEC_IODRV.IoDrvModes.IODRV_MODE_DI_ENABLED);
END_IF

IF result = EPEC_SYSTEM.SYSTEM_ERROR_CODES.FW_ERR_OK THEN
	connector := 255; // internal
	pin := 1;
	result := EPEC_IODRV.IoDrvDISetMode(EPEC_HW.IO_Channels.PIN_1000_1_DI_SERVICE_MODE, EPEC_IODRV.IoDrvModes.IODRV_MODE_DI_ENABLED);
END_IF

IF result = EPEC_SYSTEM.SYSTEM_ERROR_CODES.FW_ERR_OK THEN
	connector := 255; // internal
	pin := 1;
	result := EPEC_IODRV.IoDrvAISetMode(EPEC_HW.IO_Channels.PIN_1000_1_AI_PCB1_Temp, EPEC_IODRV.IoDrvModes.IODRV_MODE_AI_ENABLED);
END_IF

IF result = EPEC_SYSTEM.SYSTEM_ERROR_CODES.FW_ERR_OK THEN
	connector := 255; // internal
	pin := 1;
	result := EPEC_IODRV.IoDrvAISetMode(EPEC_HW.IO_Channels.PIN_1000_1_AI_PCB2_Temp, EPEC_IODRV.IoDrvModes.IODRV_MODE_AI_ENABLED);
END_IF

IF result = EPEC_SYSTEM.SYSTEM_ERROR_CODES.FW_ERR_OK THEN
	connector := 255; // internal
	pin := 1;
	result := EPEC_IODRV.IoDrvAISetMode(EPEC_HW.IO_Channels.PIN_1000_1_AI_MCU_Temp, EPEC_IODRV.IoDrvModes.IODRV_MODE_AI_ENABLED);
END_IF

IF result = EPEC_SYSTEM.SYSTEM_ERROR_CODES.FW_ERR_OK THEN
	connector := 255; // internal
	pin := 1;
	result := EPEC_IODRV.IoDrvAISetMode(EPEC_HW.IO_Channels.PIN_1000_1_AI_SBC_Temp, EPEC_IODRV.IoDrvModes.IODRV_MODE_AI_ENABLED);
END_IF

IF result = EPEC_SYSTEM.SYSTEM_ERROR_CODES.FW_ERR_OK THEN
	connector := 255; // internal
	pin := 1;
	result := EPEC_IODRV.IoDrvAISetMode(EPEC_HW.IO_Channels.PIN_1000_1_AI_VIN_M, EPEC_IODRV.IoDrvModes.IODRV_MODE_AI_ENABLED);
END_IF

IF result = EPEC_SYSTEM.SYSTEM_ERROR_CODES.FW_ERR_OK THEN
	connector := 255; // internal
	pin := 1;
	result := EPEC_IODRV.IoDrvAISetMode(EPEC_HW.IO_Channels.PIN_1000_1_AI_VOUT_SAFE_M, EPEC_IODRV.IoDrvModes.IODRV_MODE_AI_ENABLED);
END_IF

IF result = EPEC_SYSTEM.SYSTEM_ERROR_CODES.FW_ERR_OK THEN
	connector := 255; // internal
	pin := 1;
	result := EPEC_IODRV.IoDrvAISetMode(EPEC_HW.IO_Channels.PIN_1000_1_AI_VOUT_NON_SAFE_M, EPEC_IODRV.IoDrvModes.IODRV_MODE_AI_ENABLED);
END_IF

IF result = EPEC_SYSTEM.SYSTEM_ERROR_CODES.FW_ERR_OK THEN
	connector := 255; // internal
	pin := 1;
	result := EPEC_IODRV.IoDrvAISetMode(EPEC_HW.IO_Channels.PIN_1000_1_AI_BSL_VOLT, EPEC_IODRV.IoDrvModes.IODRV_MODE_AI_ENABLED);
END_IF
  
IF result = EPEC_SYSTEM.SYSTEM_ERROR_CODES.FW_ERR_OK THEN
	result := EPEC_IODRV.IoDrvSetState(EPEC_IODRV.IoDrvStates.IODRV_STATE_RUN);
	o_FWErrorCode := result;
END_IF

IF result <> EPEC_SYSTEM.SYSTEM_ERROR_CODES.FW_ERR_OK THEN
	o_Error:=TRUE;
	o_ErrorInConnector := connector;
	o_ErrorInPin := pin;
	o_FWErrorCode := result;

	info1:= SHL(connector, 16) OR pin;
	EPEC_SERRLOG.S_AddError_DWORD(
		i_ErrorCode:= ApplicationErrors.IO_INIT,
		i_LibraryErrorCode:= result,
		i_Info1:= info1, // MSW connector, LSW pin
		i_Info2:= info2 // error specific
	);
END_IF

o_Ready:=TRUE;

          
END_PROGRAM

(* NOTE! NOTE! NOTE! NOTE! NOTE! NOTE! NOTE! NOTE! NOTE! NOTE! NOTE! This object is created by Epec MultiTool User changes are overwritten when project is imported Content(input conversion, validation and diagnostic): - Validate all safe inputs using * S_ADCToVoltageOrCurrent() * S_ValidateAI() * S_VoltageToDI() * S_ValidateDI() * S_AIOverCurrentProtection(). All FB's o_Status.OutputValid output statuses will be taken in count into 'inputs valid' status. This PRG contains safety-related code. The following attribute is autogenerated. Do not remove. *)
{attribute 'hide_all_locals'}
{attribute 'analysis' := '-3, -9, -29, -33, -35, -130'}
PROGRAM S_Inputs
  VAR_INPUT
    i_Enable : BOOL := TRUE;
    i_Initialize : BOOL := TRUE;
  END_VAR
  VAR_OUTPUT
    o_InitReady : BOOL := FALSE;
    o_AI_VIN_V_Diagnostic : DWORD;  (* Filtered ADC value for supply voltage (VIN_M) *)
    o_AI_PCB_1_V_Diagnostic : DWORD;  (* Filtered ADC value for PCB1 temperature *)
    o_AI_PCB_2_V_Diagnostic : DWORD;  (* Filtered ADC value for PCB2 temperature *)
    o_AI_MCU_C_Diagnostic : DINT;  (* MCU temperature [0.1 C] *)
    o_AI_SBC_C_Diagnostic : DINT;  (* SBC temperature [0.1 C] *)
    o_AI_VOUT_SAFE_Diagnostic : DWORD;  (* Filtered ADC value for voltage after safety switch (VOUT_SAFE_M) *)
    o_AI_VOUT_NON_SAFE_Diagnostic : DWORD;  (* Filtered ADC value for voltage before safety switch (VOUT_NONSAFE_M) *)
    o_AI_BSL_V_Diagnostic : DWORD;  (* Filtered ADC value for BSL voltage *)
    o_DI_FACTORY_RESET_Diagnostic : BYTE;  (* Factory reset state *)
    o_DI_SERVICE_MODE_Diagnostic : BYTE;  (* Service mode state *)
    o_UptimeWarning_Diagnostic : BOOL;  (* Uptime warning, maximum runtime approaching *)
    o_UptimeExceeded_Diagnostic : BOOL;  (* Uptime exceeded, runtime after bootup over limit *)
    o_Uptime_Elapsed_Diagnostic : TIME;  (* Elapsed time since bootup, counts up to the allowed 24h *)
  END_VAR
  VAR
    AI_VIN_V_Diagnostic : DWORD;  (* Internal diagnostic variable mapped to FW io interface *)
    AI_PCB_1_V_Diagnostic : DWORD;  (* Internal diagnostic variable mapped to FW io interface *)
    AI_PCB_2_V_Diagnostic : DWORD;  (* Internal diagnostic variable mapped to FW io interface *)
    AI_MCU_C_Diagnostic : DINT;  (* Internal diagnostic variable mapped to FW io interface *)
    AI_SBC_C_Diagnostic : DINT;  (* Internal diagnostic variable mapped to FW io interface *)
    AI_VOUT_SAFE_Diagnostic : DWORD;  (* Internal diagnostic variable mapped to FW io interface *)
    AI_VOUT_NON_SAFE_Diagnostic : DWORD;  (* Internal diagnostic variable mapped to FW io interface *)
    AI_BSL_V_Diagnostic : DWORD;  (* Internal diagnostic variable mapped to FW io interface *)
    DI_FACTORY_RESET_Diagnostic : BYTE;  (* Internal diagnostic variable mapped to FW io interface *)
    DI_SERVICE_MODE_Diagnostic : BYTE;  (* Internal diagnostic variable mapped to FW io interface *)
    uptimeWarningTimer_Diagnostic : Standard.TON;  (* TON timer for uptime warning *)
    uptimeExceededTimer_Diagnostic : Standard.TON;  (* TON timer for uptime exceeded *)
  END_VAR

            IF(i_Initialize) THEN
	o_InitReady:= TRUE;
  
ELSE

	(* Copy measured diagnostic signals to outputs *)
	o_AI_VIN_V_Diagnostic := AI_VIN_V_Diagnostic;
	o_AI_VOUT_SAFE_Diagnostic := AI_VOUT_SAFE_Diagnostic;
	o_AI_VOUT_NON_SAFE_Diagnostic := AI_VOUT_NON_SAFE_Diagnostic;

	o_AI_BSL_V_Diagnostic := AI_BSL_V_Diagnostic;
	o_DI_FACTORY_RESET_Diagnostic := DI_FACTORY_RESET_Diagnostic;
	o_DI_SERVICE_MODE_Diagnostic := DI_SERVICE_MODE_Diagnostic;

 	o_AI_MCU_C_Diagnostic := AI_MCU_C_Diagnostic;
	o_AI_SBC_C_Diagnostic := AI_SBC_C_Diagnostic;
	o_AI_PCB_1_V_Diagnostic := AI_PCB_1_V_Diagnostic;
	o_AI_PCB_2_V_Diagnostic := AI_PCB_2_V_Diagnostic;

	uptimeWarningTimer_Diagnostic(
		IN:=TRUE,
		PT:=T#23H30M,
		Q=>o_UptimeWarning_Diagnostic,
		ET=>
	);

	uptimeExceededTimer_Diagnostic(
		IN:=TRUE,
		PT:=T#24H,
		Q=>o_UptimeExceeded_Diagnostic,
		ET=> o_Uptime_Elapsed_Diagnostic
	);



  
END_IF

          
END_PROGRAM

(* NOTE! NOTE! NOTE! NOTE! NOTE! NOTE! NOTE! NOTE! NOTE! NOTE! NOTE! This object is created by Epec MultiTool User changes are overwritten when project is imported Content - Init and update all used SafeSSeriesDiagnostic library FB instances * S_DOControlAndDiagnostics() * S_DOValveEcoControlAndDiagnostics() All Init methods return TRUE if ok. They will be taken in count into Ready status. This PRG contains non safety-related code. The following attribute is autogenerated. Do not remove. *)
{attribute 'hide_all_locals'}
{attribute 'analysis' := '-3, -9, -29, -33, -35, -130'}
PROGRAM S_Outputs
  VAR_INPUT
    i_Enable : BOOL := TRUE;
    i_Initialize : BOOL := TRUE;
    i_UpdateMeasurements : BOOL := FALSE;
  END_VAR
  VAR_OUTPUT
    o_InitReady : BOOL := FALSE;
    o_TotalOutputCurrent_Diagnostic : DINT;  (* Sum of all output current measurements *)
  END_VAR
  VAR
    TotalOutputCurrent_Diagnostic : DINT;  (* Sum of all output current measurements *)
    pin : DWORD := DWORD#0;
    connector : DWORD := DWORD#0;
    info1 : DWORD := DWORD#0;
    info2 : DWORD := DWORD#0;
    errorCode : DINT := DINT#0;
  END_VAR

            IF(i_Initialize) THEN
	o_InitReady:= TRUE;
  
ELSIF i_UpdateMeasurements THEN
  
;
ELSE

	(* Copy measured diagnostic signals to outputs *)
	o_TotalOutputCurrent_Diagnostic := TotalOutputCurrent_Diagnostic;



  
END_IF

          
END_PROGRAM
